SUPER^();
M_mapping();
IF sInstanceName='tote_1' THEN
	tote_status_array[0]	:= GVL.fb_loading.tote_status;
	tote_status_array[1]	:= GVL.fb_working1.tote_status;
	tote_status_array[2]	:= GVL.fb_working1.outboundTote_status;//outbound tote status form logtech
	machine_current_status	:= GVL.PackTags1.Status.StateCurrent;
	autostore_status		:= GVL.fb_autoStore1.autostore_status;
END_IF
IF sInstanceName='tote_2' THEN
	tote_status_array[0]	:= GVL.fb_loading.tote_status;
	tote_status_array[1]	:= GVL.fb_working2.tote_status;
	tote_status_array[2]	:= GVL.fb_working2.outboundTote_status;//outbound tote status form logtech
	machine_current_status	:= GVL.PackTags2.Status.StateCurrent;
	autostore_status		:= GVL.fb_autoStore2.autostore_status;
END_IF

CASE machine_current_status OF
	ePMLState_Aborted,ePMLState_Aborting:
		status	:= MachineStatus.ERROR;
	ePMLState_Stopping:	
		status	:= MachineStatus.STOPPING;
	ePMLState_Stopped:
		status	:= MachineStatus.STOPPED;
	ePMLState_Resetting:	
		status	:= MachineStatus.RESETTING;
	ePMLState_Idle:	
		status	:= MachineStatus.READY;		
	ePMLState_Execute:	
		status	:= MachineStatus.RUNNING;			
END_CASE

IF bInbound THEN
	inboundToteParams_temp.source_id	:= ModelIdentifier.inbounding_position;
	inboundToteParams_temp.target_id	:= ModelIdentifier.working_position;
	inbound_tote_request(inbound_tote_params:=inboundToteParams_temp);
	bInbound	:= FALSE;
END_IF
IF bOutbound THEN
	outboundToteParams_temp.source_id	:= ModelIdentifier.working_position;
	outboundToteParams_temp.target_id	:= ModelIdentifier.outbound_position;	
	outbound_tote_request(outbound_tote_params:=outboundToteParams_temp);
	bOutbound	:= FALSE;
END_IF
IF bAbortInbound THEN
	abortToreParams_temp.source_id	:= ModelIdentifier.inbounding_position;
	abortToreParams_temp.target_id	:= ModelIdentifier.working_position;	
	abort_tote_request(abort_tote_request_params:=abortToreParams_temp);
	bAbortInbound	:= FALSE;
END_IF

IF bAbortOutbound THEN
	abortToreParams_temp.source_id	:= ModelIdentifier.working_position;
	abortToreParams_temp.target_id	:= ModelIdentifier.outbound_position;	
	abort_tote_request(abort_tote_request_params:=abortToreParams_temp);
	bAbortOutbound	:= FALSE;
END_IF
IF bAutostore_exchange THEN
	autostore_control_command(Command:=AutostoreControlCommand.START);
	bAutostore_exchange	:= FALSE;
END_IF

{attribute 'TcRpcEnable'}
METHOD abort_tote_request : UDINT//only response while awaiting
VAR_INPUT
	abort_tote_request_params : AbortToteRequestParams; // Struct containing data from the barcode scan	
END_VAR
abort_tote_request:=MethodCallReturnValue.DECLINED_BUSY;
IF sInstanceName='tote_1' THEN
	IF abort_tote_request_params.source_id=ModelIdentifier.inbounding_position AND abort_tote_request_params.target_id=ModelIdentifier.working_position THEN
		iCase_abort	:= 1;
	END_IF
	IF abort_tote_request_params.source_id=ModelIdentifier.working_position AND abort_tote_request_params.target_id=ModelIdentifier.outbound_position THEN
		iCase_abort	:= 2;
	END_IF		
	CASE iCase_abort OF
		1:
			IF GVL.fb_working1.tote_status=ToteStatus.AWAITING_INBOUND_AVAILABILITY THEN
				subData.Topic	:= E_Topics.WORKING1_ABORT_INBOUND;
				GVL.PubSubService.Publish(topic:=E_Topics.WORKING1_ABORT_INBOUND,data:= subData);
				abort_tote_request:= MethodCallReturnValue.ACCEPTED;
			ELSE
				abort_tote_request:= MethodCallReturnValue.DECLINED_ERROR;
			END_IF
		2:
			IF GVL.fb_working1.tote_status=ToteStatus.AWAITING_OUTBOUND_AVAILABILITY THEN
				subData.Topic	:= E_Topics.WORKING1_ABORT_OUTBOUND;
				GVL.PubSubService.Publish(topic:=E_Topics.WORKING1_ABORT_OUTBOUND,data:= subData);
				abort_tote_request:= MethodCallReturnValue.ACCEPTED;
			ELSE
				abort_tote_request:= MethodCallReturnValue.DECLINED_ERROR;
			END_IF	
		ELSE
			abort_tote_request:= MethodCallReturnValue.DECLINED_ERROR;
	END_CASE
END_IF

IF sInstanceName='tote_2' THEN
	IF abort_tote_request_params.source_id=ModelIdentifier.inbounding_position AND abort_tote_request_params.target_id=ModelIdentifier.working_position THEN
		iCase_abort	:= 1;
	END_IF
	IF abort_tote_request_params.source_id=ModelIdentifier.working_position AND abort_tote_request_params.target_id=ModelIdentifier.outbound_position THEN
		iCase_abort	:= 2;
	END_IF		
	CASE iCase_abort OF
		1:
			IF GVL.fb_working2.tote_status=ToteStatus.AWAITING_INBOUND_AVAILABILITY THEN
				subData.Topic	:= E_Topics.WORKING2_ABORT_INBOUND;
				GVL.PubSubService.Publish(topic:=E_Topics.WORKING2_ABORT_INBOUND,data:= subData);
				abort_tote_request:= MethodCallReturnValue.ACCEPTED;
			ELSE
				abort_tote_request:= MethodCallReturnValue.DECLINED_ERROR;
			END_IF
		2:
			IF GVL.fb_working2.tote_status=ToteStatus.AWAITING_INBOUND_AVAILABILITY THEN
				subData.Topic	:= E_Topics.WORKING2_ABORT_OUTBOUND;
				GVL.PubSubService.Publish(topic:=E_Topics.WORKING2_ABORT_OUTBOUND,data:= subData);
				abort_tote_request:= MethodCallReturnValue.ACCEPTED;
			ELSE
				abort_tote_request:= MethodCallReturnValue.DECLINED_ERROR;
			END_IF	
		ELSE
			abort_tote_request:= MethodCallReturnValue.DECLINED_ERROR;			
	END_CASE
END_IF
END_METHOD

{attribute 'TcRpcEnable'}
METHOD autostore_control_command : BOOL
VAR_INPUT
	Command	: AutostoreControlCommand;
END_VAR
autostore_control_command	:= FALSE;
IF sInstanceName='tote_1' THEN
	subData.Topic	:= E_Topics.AUTOSTORE1_EXCHANGE;
	GVL.PubSubService.Publish(topic:= E_Topics.AUTOSTORE1_EXCHANGE,data:= subData);
END_IF
IF sInstanceName='tote_2' THEN
	subData.Topic	:= E_Topics.AUTOSTORE2_EXCHANGE;
	GVL.PubSubService.Publish(topic:= E_Topics.AUTOSTORE2_EXCHANGE,data:= subData);
END_IF
autostore_control_command	:= TRUE;
END_METHOD

{attribute 'TcRpcEnable'}
METHOD barcode_validation_request : UDINT
VAR_INPUT
	barcode_validation_request_params : BarcodeValidationRequestParams;
END_VAR
END_METHOD

{attribute 'TcRpcEnable'}
METHOD inbound_tote_request : UDINT
VAR_INPUT
	inbound_tote_params : InboundToteParams;
END_VAR
VAR	
	subData	: PubSubData;
END_VAR

IF sInstanceName='tote_1' THEN
//	IF NOT (((GVL.fb_working1.xLoading OR GVL.fb_working1.xInbound) AND GVL.fb_loading.xOutbound_woking1) OR 
//		GVL.fb_working1.tote_status=ToteStatus.LOADED OR GVL.fb_working1.xUnloading OR GVL.fb_working1.xOutbound) 
//	THEN//avoid cmd while inbounding or has tote
//		subData.Topic	:= E_Topics.WORKING1_INBOUND_TOTE;
//		GVL.PubSubService.Publish(topic:= E_Topics.WORKING1_INBOUND_TOTE,data:= subData);	
//	END_IF
	subData.Topic	:= E_Topics.WORKING1_INBOUND_TOTE;
	GVL.PubSubService.Publish(topic:= E_Topics.WORKING1_INBOUND_TOTE,data:= subData);
	A1	:= A1+1;	
END_IF
IF sInstanceName='tote_2' THEN
//	IF NOT (((GVL.fb_working2.xLoading OR GVL.fb_working2.xInbound) AND GVL.fb_loading.xOutbound_woking2) OR 
//		GVL.fb_working2.tote_status=ToteStatus.LOADED OR GVL.fb_working2.xUnloading OR GVL.fb_working2.xOutbound) 
//	THEN//avoid cmd while inbounding or has tote
//		subData.Topic	:= E_Topics.WORKING2_INBOUND_TOTE;
//		GVL.PubSubService.Publish(topic:= E_Topics.WORKING2_INBOUND_TOTE,data:= subData);
//	END_IF
	subData.Topic	:= E_Topics.WORKING2_INBOUND_TOTE;
	GVL.PubSubService.Publish(topic:= E_Topics.WORKING2_INBOUND_TOTE,data:= subData);
	A2	:= A2+1;
END_IF

//subData.Topic	:= E_Topics.RESET_WAITING_FOR_NEW_SPACE;
//GVL.PubSubService.Publish(topic:= E_Topics.RESET_WAITING_FOR_NEW_SPACE,data:= subData);
END_METHOD

{attribute 'TcRpcEnable'}
METHOD  init_tote_request : udint
VAR_INPUT
	init_tote_request_params : InitToteRequestParams;
END_VAR
init_tote_request:=1;
IF init_tote_request_params.source_id=ModelIdentifier.inbounding_position AND 
   init_tote_request_params.source_id=ModelIdentifier.working_position THEN 
  ;
     //MAIN.Machine.EM03.eState:=	E_WorkingStates.IDLE;				
//			MAIN.Machine.EM03.xLoading	:= FALSE;
//			MAIN.Machine.EM03.xUnloading	:= FALSE;
//			MAIN.Machine.EM03.xPerturbing := FALSE;
//			MAIN.Machine.EM03.xSwaping    := FALSE;
	 //MAIN.Machine.EM01.eState:=E_LoadingStates.IDLE;
END_IF  
IF init_tote_request_params.source_id=ModelIdentifier.working_position AND 
   init_tote_request_params.source_id=ModelIdentifier.outbound_position THEN 
;
    // MAIN.Machine.EM03.eState:=	E_WorkingStates.IDLE;				
//			MAIN.Machine.EM03.xLoading	:= FALSE;
//			MAIN.Machine.EM03.xUnloading	:= FALSE;
//			MAIN.Machine.EM03.xPerturbing := FALSE;
//			MAIN.Machine.EM03.xSwaping    := FALSE;
	// MAIN.Machine.EM04.eState:=E_UnloadingStates.IDLE;
END_IF  
init_tote_request:=0;
END_METHOD

METHOD M_mapping : BOOL
VAR_INPUT
END_VAR
END_METHOD

{attribute 'TcRpcEnable'}
METHOD outbound_tote_request : UDINT
VAR_INPUT
	outbound_tote_params : OutboundToteParams;	
END_VAR
VAR	
	subData	: PubSubData;
END_VAR
IF sInstanceName='tote_1' THEN
	IF NOT (GVL.fb_working1.xOutbound OR GVL.fb_working1.xInbound ) THEN//avoid cmd while outbounding
		subData.Topic	:= E_Topics.WORKING1_OUTBOUND_TOTE;
		GVL.PubSubService.Publish(topic:= E_Topics.WORKING1_OUTBOUND_TOTE,data:= subData);
	END_IF	
END_IF
IF sInstanceName='tote_2' THEN
	IF NOT (GVL.fb_working2.xOutbound OR GVL.fb_working2.xInbound ) THEN//avoid cmd while outbounding
		subData.Topic	:= E_Topics.WORKING2_OUTBOUND_TOTE;
		GVL.PubSubService.Publish(topic:= E_Topics.WORKING2_OUTBOUND_TOTE,data:= subData);
	END_IF
END_IF
END_METHOD

{attribute 'TcRpcEnable'}
METHOD perturb_tote_request : UDINT
VAR_INPUT
	perturb_tote_params : PerturbToteParams;	
END_VAR
IF //APP.Machine.CurrentStateEnum=E_PMLState.ePMLState_Execute 
//AND 
cmd=OrderToteCommand.DO_NOTHING
AND NOT MAIN.safety_1.bStop_button_unlock 
//AND NOT MAIN.safety_1.bBStop_button_unlock 
THEN
	cmd	:= OrderToteCommand.OPEN_BAG;
	perturb_tote_request:=0;
ELSE
	perturb_tote_request:=1;
END_IF
END_METHOD

{attribute 'TcRpcEnable'}
METHOD reset_tote_request : UDINT
VAR_INPUT
		
END_VAR
reset_tote_request	:= 1;

GVL.PackTags.Command.CntrlCmd:=1;

reset_tote_request	:= 0;
END_METHOD

{attribute 'TcRpcEnable'}
METHOD Setcmd : BOOL
VAR_INPUT
	orderToteCommand : OrderToteCommand;
END_VAR
cmd	:= orderToteCommand;
END_METHOD

{attribute 'TcRpcEnable'}
METHOD swap_tote_request : UDINT
VAR_INPUT
	swap_tote_params : SwapToteParams;	
END_VAR
IF //APP.Machine.CurrentStateEnum=E_PMLState.ePMLState_Execute 
//AND 
cmd=OrderToteCommand.DO_NOTHING
AND NOT MAIN.safety_1.bStop_button_unlock 
//AND NOT MAIN.safety_1.bBStop_button_unlock 
THEN
	cmd	:= OrderToteCommand.SWAP;
	swap_tote_request:=0;
ELSE
	swap_tote_request:=1;
END_IF
END_METHOD

END_FUNCTION_BLOCK

// ---- Mian/MAIN.TcPOU
// Disclaimer
// 
// This publication contains statements about the suitability of our products for certain areas of application. These statements are based on typical features of our products. The examples shown in this publication are for demonstration purposes only. 
// The information provided herein should not be regarded as specific operation characteristics. It is incumbent on the customer to check and decide whether a product is suitable for use in a particular application. 
// We do not give any warranty that the source code which is made available with this publication is complete or accurate. 
//
// THE SAMPLE CODE CONTAINED IN THIS PUBLICATION IS PROVIDED “AS IS” WITHOUT WARRANTY OF ANY KIND, EITHER EXPRESSED, IMPLIED OR STATUTORY, INCLUDING WITHOUT LIMITATION, ANY WARRANTY WITH RESPECT TO NON-INFRINGEMENT, FREEDOM FROM PROPRIETARY RIGHTS OF THIRD PARTIES OR FITNESS FOR ANY PARTICULAR PURPOSE. 
// This publication may be changed from time to time without prior notice. No liability is assumed for errors and/or omissions. Our products are described in detail in our data sheets and documentations. Product-specific warnings and cautions must be observed. 
// For the latest version of our data sheets and documentations visit our website (www.beckhoff.de). 
//
// © Beckhoff Automation GmbH & Co. KG, 2022
// The reproduction, distribution and utilization of this document as well as the communication of its contents to others without express authorization is prohibited. Offenders will be held liable for the payment of damages. All rights reserved in the event of the grant of a patent, utility model or design.
PROGRAM MAIN
VAR_INPUT
	bExecuteComplete			: BOOL;									//Command Execute Complete, not defined
END_VAR
VAR
	firstCycle : BOOL := TRUE;
	UserModeCofig				: PML_UnitModeConfig;					//User can configure his own Mode
	
	fbMachine					: FB_Machine;							//Instance of FB_Machine
//	fbMachine_2					: FB_Machine;							//Instance of FB_Machine
	bMachineStartedUp			: BOOL := FALSE;						//TRUE, when first PLC-Cycle finish
	fbVisu						: FB_Visu;								//Visualization
							//Visualization
	fbTrigger					: F_TRIG;								//Trigger for resseting Counters
	fbTrigger_2					: F_TRIG;								//Trigger for resseting Counters

	fbLocalSystemTime			 : FB_LocalSystemTime;					//Get local Systemtime
	fbLocalSystemTime_2			 : FB_LocalSystemTime;					//Get local Systemtime
	
	fbTriggerErrorMainAxis		: R_TRIG;								//Trigger for detecting Error on Mainaxis and write into PackTags
	fbTriggerErrorMetalAxis		: R_TRIG;								//Trigger for detecting Error on Metalaxis and write into PackTags
	fbTriggerErrorPlasticAxis	: R_TRIG;								//Trigger for detecting Error on Plasticaxis and write into PackTags
	
	nStateCommandCheck			: DINT;									//State to handle with statecommands
	
	i	: INT;

	FB_GetUPSStatus: FB_GetUPSStatus;	
	dataloaded: BOOL;								//UPS数据文件读取状态（True为读取成功，False为读取失败）
	OldData: BOOL;									//UPS备份数据文件读取状态
	PersistentDataStatus: EPlcPersistentStatus;		//Persistent数据读取（恢复）状态	
//	fb_ups	:FB_S_UPS_CX51x0;
	//application	: FB_Application;

	bButton				: BOOL;
	ton_button			: TON;

	refMachine_control_cmd	:REFERENCE TO MachineControlCommand;
	
	refMachine_control_cmd_2	:REFERENCE TO MachineControlCommand;
	
	rTrig_error	:ARRAY[0..10] OF R_TRIG;
	rTrig_error_2	:ARRAY[0..10] OF R_TRIG;
	
	rTrig_agingTest	:R_TRIG;
	fTrig_agingTest	:F_TRIG;

	topicCallbackTest	: E_Topics;
	dataCallbackTest	: PubSubData;
	topic_sample	: E_topic_sample;
	
	(***********************ADS********************************)
	light_tower_1			:	FB_Light_tower_module;
	light_tower_2			:	FB_Light_tower_module;
   // application_1			:	FB_Application;
	tote_1					:	FB_Tote_Subsystem;
	tote_2					:	FB_Tote_Subsystem;
	safety_1				:	FB_Safety_Subsystem;
	safety_2				:	FB_Safety_Subsystem;
	machine_control_1		:	FB_MachineControl_Subsystem;
	machine_control_2		:	FB_MachineControl_Subsystem;
	heartbeat_1				:	FB_HeartBeat_Subsystem;
	heartbeat_2				:	FB_HeartBeat_Subsystem;
	
	air_pressure_1			:	FB_AirPressure_Subsystem;
	air_pressure_2			:	FB_AirPressure_Subsystem;
	
	
	heartbeat_data_test : HeartbeatParams;	
	update_light_tower_params_test	: UpdateLightTowerParams;
	tset1: UDINT;
	
	
	version 				:	STRING(255);
	testbool: BOOL;
	inbound_tote_params_test : InboundToteParams;
	OutboundToteParams_test		:	OutboundToteParams;
	testbool1: BOOL;
	
	
	
	fbMachine1					: FB_Machine;							//Instance of FB_Machine
	fbMachine2					: FB_Machine;							//Instance of FB_Machine
	stateMachine1	: FB_StateMachine;
	stateMachine2	: FB_StateMachine;
	
	
END_VAR

(**************************************UPS*****************************************)
FB_GetUPSStatus(
	sNetId:= , 					//默认为本机Netid
	nPort:= , 					//ADS端口号，若不填写功能块会自动获取，默认0
	bEnable:= , 				//高电平有效，置True后循环读取UPS状态
	bValid=> , 					//当bValid为True时，stStatus的值有效
	bError=> , 
	nErrId=> , 
	stStatus=> );				//包含UPS信息的结构体
	

dataloaded:=_Appinfo.BootDataLoaded;
OldData:=_Appinfo.OldBootData;
PersistentDataStatus:=_Appinfo.PersistentStatus;

//application();
version:='v1.0.0';


//Call FB_Machine

GVL.fb_loading();
GVL.fb_working1();
GVL.fb_working2();
GVL.fb_autoStore1();
GVL.fb_autoStore2();
GVL.fb_working1._iModuleID:= ModuleID.WORKING1;
GVL.fb_working1._sInstanceName	:= 'working1';
GVL.fb_loading._iModuleID:= ModuleID.LOADING;
GVL.fb_loading._sInstanceName	:= 'loading';
GVL.fb_working2._iModuleID:= ModuleID.WORKING2;
GVL.fb_working2._sInstanceName	:= 'working2';
GVL.fb_autoStore1._sInstanceName	:= 'autoStore_1';
GVL.fb_autoStore1._iModuleID	:= ModuleID.AUTOSTORE1;
GVL.fb_autoStore2._sInstanceName	:= 'autoStore_2';
GVL.fb_autoStore2._iModuleID	:= ModuleID.AUTOSTORE2;

(***********************ADS********************************)
GVL.fb_mcp_1(id:=1);
heartbeat_1();
air_pressure_1(pPackTags:=ADR(GVL.PackTags1));
machine_control_1(pMachineCurrentStatus:= ADR(GVL.PackTags1.Status.StateCurrent));
tote_1();
safety_1(pHeartBeat:=ADR(heartbeat_1),pSafety_door:=ADR(GVL.fb_mcp_1.st_safety_door),pPackTags:=ADR(GVL.PackTags1),pMachine:=ADR(fbMachine1));
light_tower_1(pHeartBeat:=ADR(heartbeat_1),pLightTower:= ADR(GVL.fb_mcp_1.lightTower));

heartbeat_1._sInstanceName	:= 'heartBeat_1';
tote_1._sInstanceName	:='tote_1';
safety_1._sInstanceName	:='safety_1';
air_pressure_1._sInstanceName	:='air_pressure1';



GVL.fb_mcp_2(id:=2);
heartbeat_2();
air_pressure_2(pPackTags:=ADR(GVL.PackTags2));
machine_control_2(pMachineCurrentStatus:= ADR(GVL.PackTags2.Status.StateCurrent));
tote_2();
light_tower_2(pHeartBeat:=ADR(heartbeat_2),pLightTower:= ADR(GVL.fb_mcp_2.lightTower));
safety_2(pHeartBeat:=ADR(heartbeat_2),pSafety_door:=ADR(GVL.fb_mcp_2.st_safety_door),pPackTags:=ADR(GVL.PackTags2),pMachine:=ADR(fbMachine2));

heartbeat_1._sInstanceName	:= 'heartBeat_2';
tote_2._sInstanceName	:='tote_2';
safety_2._sInstanceName	:='safety_2';
air_pressure_2._sInstanceName	:='air_pressure2';





//Configure Usermode 1
A_UnitModeConfig();

//Runs the first PLC-Cycle
IF fbMachine1.bUndefinedDone AND fbMachine2.bUndefinedDone AND NOT bMachineStartedUp THEN
	GVL.PackTags1.Command.CntrlCmd	:= ePMLCommand_Abort;
	GVL.PackTags2.Command.CntrlCmd	:= ePMLCommand_Abort;
	bMachineStartedUp			:= TRUE;
END_IF


GVL.bButtonProductionReq := GVL.PackTags.Command.UnitMode = ePMLProtUnitMode_Production AND GVL.PackTags.Status.UnitModeCurrent <> GVL.PackTags.Command.UnitMode;

//Set the Packtags
M_SetPackTags();

//set the errors and warnings in Packtags
M_SetPackTagsErrorWarning();

//Call Visu
M_CallVisu();
///////////////////initialize unitmode and set 
IF GVL.PackTags.Command.UnitMode=ePMLProtUnitMode_Invalid THEN
	GVL.PackTags.Command.UnitMode	:= ePMLProtUnitMode_Production;
	GVL.PackTags.Command.Parameter[1].Value := 1;
	GVL.PackTags1.Command.UnitMode	:= ePMLProtUnitMode_Production;
	GVL.PackTags1.Command.Parameter[1].Value := 1;	
	GVL.PackTags2.Command.UnitMode	:= ePMLProtUnitMode_Production;
	GVL.PackTags2.Command.Parameter[1].Value := 1;	
	
END_IF


fbMachine1(	eModeCommand:= GVL.PackTags.Command.UnitMode,
  			eMode => GVL.PackTags1.Status.UnitModeCurrent, 
			eState =>GVL.PackTags1.Status.StateCurrent,
			pPML_Instance1:=ADR(GVL.fb_working1),
			pPML_Instance2:=ADR(GVL.fb_loading),
			pPackTags:=ADR(GVL.PackTags1),
			pSafetySystem	:= ADR(safety_1)
			);
			
fbMachine2(	eModeCommand:= GVL.PackTags.Command.UnitMode,
  			eMode => GVL.PackTags2.Status.UnitModeCurrent, 
			eState =>GVL.PackTags2.Status.StateCurrent,
			pPML_Instance1:=ADR(GVL.fb_working2),
			pPML_Instance2:=ADR(GVL.fb_loading),
			pPackTags:=ADR(GVL.PackTags2),
			pSafetySystem	:= ADR(safety_2)
			);		
	
stateMachine1(	pPackTags:=ADR(GVL.PackTags1),
				pMachine:=ADR(fbMachine1),
				pMachine_control_cmd := ADR(machine_control_1.machineControlCmd),
				pAirSystem	:=ADR(air_pressure_1),
				pSafetySystem	:= ADR(safety_1),
				pMcp	:= ADR(GVL.fb_mcp_1)
				);

stateMachine2(	pPackTags:=ADR(GVL.PackTags2),
				pMachine:=ADR(fbMachine2),
				pMachine_control_cmd := ADR(machine_control_2.machineControlCmd),
				pAirSystem	:=ADR(air_pressure_2),
				pSafetySystem	:= ADR(safety_2),
				pMcp	:= ADR(GVL.fb_mcp_2)
				);			
		
			
GVL.fbWriteLog(
	bWrite:= GVL.bWrite, 
	sFileName:= , 
	sMessage:= , 
	OK=> , 
	Busy=> , 
	ErrorMsg=> , 
	bError=> , 
	ErrorID=> );
	



M_SetUnitInfo();

ACTION A_UnitModeConfig:
UserModeCofig(
	eMode							:= ePMLUnitMode_Service, 
	bDisableClearing				:= TRUE, 
	bDisableStarting				:= FALSE, 
	bDisableSuspended				:= FALSE, 
	bDisableStopping				:= TRUE, 
	bDisableAborting				:= TRUE, 
	bDisableHolding					:= TRUE, 
	bDisableHeld					:= TRUE, 
	bDisableUnholding				:= TRUE, 
	bDisableSuspending				:= TRUE, 
	bDisableUnsuspending			:= TRUE, 
	bDisableResetting				:= TRUE, 
	bDisableIdle					:= FALSE, 
	bDisableCompleting				:= TRUE, 
	bDisableComplete				:= FALSE, 
	bEnableUnitModeChangeStopped	:= TRUE, 
	bEnableUnitModeChangeIdle		:= TRUE, 
	bEnableUnitModeChangeSuspended	:= FALSE, 
	bEnableUnitModeChangeExecute	:= FALSE, 
	bEnableUnitModeChangeAborted	:= TRUE, 
	bEnableUnitModeChangeHeld		:= FALSE, 
	bEnableUnitModeChangeComplete	:= TRUE, 
	bError							=> , 
	nErrorId						=> );
UserModeCofig(
	eMode							:= ePMLUnitMode_Production, 
	bDisableClearing				:= FALSE, 
	bDisableStarting				:= FALSE, 
	bDisableSuspended				:= TRUE, 
	bDisableStopping				:= FALSE, 
	bDisableAborting				:= FALSE, 
	bDisableHolding					:= TRUE, 
	bDisableHeld					:= TRUE, 
	bDisableUnholding				:= TRUE, 
	bDisableSuspending				:= TRUE, 
	bDisableUnsuspending			:= TRUE, 
	bDisableResetting				:= FALSE, 
	bDisableIdle					:= FALSE, 
	bDisableCompleting				:= FALSE, 
	bDisableComplete				:= FALSE, 
	bEnableUnitModeChangeStopped	:= TRUE, 
	bEnableUnitModeChangeIdle		:= TRUE, 
	bEnableUnitModeChangeSuspended	:= FALSE, 
	bEnableUnitModeChangeExecute	:= FALSE, 
	bEnableUnitModeChangeAborted	:= TRUE, 
	bEnableUnitModeChangeHeld		:= FALSE, 
	bEnableUnitModeChangeComplete	:= TRUE, 
	bError							=> , 
	nErrorId						=> );
END_ACTION

METHOD M_CallVisu
VAR_INPUT
END_VAR
//Calling FB_Visu
fbVisu(
	aKeyPressed				:= GVL.aKeyPressed,
	aUnitInfo				:= GVL.aUnitInfo, 
	bInvalidEntry			=> ,
	aCaption				=> GVL.aCaption,
	eModeVisu				=> ,
	eStateVisu				=> ,
	sUnitName				=> ,
	iFrameVisible			=> );
END_METHOD

METHOD M_SetPackTags
VAR_INPUT
END_VAR
VAR	
END_VAR
//***************************Writing Data into GVL.PackTags***************************

//Parameters for the production
GVL.PackTags.Command.Parameter[1].ID				:= 1;
GVL.PackTags.Command.Parameter[1].Name				:= 'Quantity';
GVL.PackTags.Command.Parameter[1].Unit				:= 'Tote';

//Countig produced totes, see fb_sample1
GVL.PackTags.Admin.ProdProcessedCount[1].ID			:= 1;
GVL.PackTags.Admin.ProdProcessedCount[1].Name		:= 'ToteFinish_Sample';
GVL.PackTags.Admin.ProdProcessedCount[1].Unit		:= 'Tote';





//Write the actual state and mode into the GVL.PackTags
GVL.PackTags.Status.StateCurrent					:= fbMachine1.eState;
GVL.PackTags.Status.UnitModeCurrent					:= fbMachine1.eMode;
GVL.PackTags.Status.StateRequested					:= fbMachine1.eCommand;
GVL.PackTags.Status.UnitModeRequested				:= fbMachine1.eModeCommand;
GVL.PackTags.Status.StateChangeInProcess			:= GVL.PackTags.Status.StateCurrent <> GVL.PackTags.Status.StateRequested;
GVL.PackTags.Status.UnitModeChangeInProcess			:= GVL.PackTags.Status.UnitModeCurrent <> GVL.PackTags.Status.UnitModeRequested;

//Write the actual state and mode into the GVL.PackTags2
GVL.PackTags1.Status.StateCurrent					:= fbMachine1.eState;
GVL.PackTags1.Status.UnitModeCurrent					:= fbMachine1.eMode;
GVL.PackTags1.Status.StateRequested					:= fbMachine1.eCommand;
GVL.PackTags1.Status.UnitModeRequested				:= fbMachine1.eModeCommand;
GVL.PackTags1.Status.StateChangeInProcess			:= GVL.PackTags1.Status.StateCurrent <> GVL.PackTags1.Status.StateRequested;
GVL.PackTags1.Status.UnitModeChangeInProcess			:= GVL.PackTags1.Status.UnitModeCurrent <> GVL.PackTags1.Status.UnitModeRequested;
//Write the actual state and mode into the GVL.PackTags2
GVL.PackTags2.Status.StateCurrent					:= fbMachine2.eState;
GVL.PackTags2.Status.UnitModeCurrent					:= fbMachine2.eMode;
GVL.PackTags2.Status.StateRequested					:= fbMachine2.eCommand;
GVL.PackTags2.Status.UnitModeRequested				:= fbMachine2.eModeCommand;
GVL.PackTags2.Status.StateChangeInProcess			:= GVL.PackTags2.Status.StateCurrent <> GVL.PackTags2.Status.StateRequested;
GVL.PackTags2.Status.UnitModeChangeInProcess			:= GVL.PackTags2.Status.UnitModeCurrent <> GVL.PackTags2.Status.UnitModeRequested;


//Write actual time and date in GVL.PackTags
fbLocalSystemTime(sNetID:= '', bEnable := TRUE);
GVL.PackTags.Admin.PlcDateTime[0]	:= fbLocalSystemTime.systemTime.wYear;
GVL.PackTags.Admin.PlcDateTime[1]	:= fbLocalSystemTime.systemTime.wMonth;
GVL.PackTags.Admin.PlcDateTime[2]	:= fbLocalSystemTime.systemTime.wDay;
GVL.PackTags.Admin.PlcDateTime[3]	:= fbLocalSystemTime.systemTime.wHour;
GVL.PackTags.Admin.PlcDateTime[4]	:= fbLocalSystemTime.systemTime.wMinute;
GVL.PackTags.Admin.PlcDateTime[5]	:= fbLocalSystemTime.systemTime.wSecond;
GVL.PackTags.Admin.PlcDateTime[6]	:= fbLocalSystemTime.systemTime.wMilliseconds;
GVL.PackTags1.Admin.PlcDateTime	:= GVL.PackTags.Admin.PlcDateTime;
GVL.PackTags2.Admin.PlcDateTime	:= GVL.PackTags.Admin.PlcDateTime;
//Set the productcounter to 0, when the production command is completed
fbTrigger(CLK:= (fbMachine1.eState = ePMLState_Complete));
IF fbTrigger.Q OR GVL.stChangeIntoProduction.bYesReset THEN
	GVL.PackTags1.Admin.ProdProcessedCount[1].Count	:= 0;
	GVL.PackTags1.Command.Parameter[1].Value			:= 0;
	GVL.nVisuProductCommand							:= 0;
END_IF

//Set the productcounter to 0, when the production command is completed
fbTrigger(CLK:= (fbMachine2.eState = ePMLState_Complete));
IF fbTrigger.Q OR GVL.stChangeIntoProduction.bYesReset THEN
	GVL.PackTags2.Admin.ProdProcessedCount[1].Count	:= 0;
	GVL.PackTags2.Command.Parameter[1].Value			:= 0;
	GVL.nVisuProductCommand							:= 0;
END_IF
END_METHOD

METHOD M_SetPackTagsErrorWarning
VAR_INPUT
END_VAR
//====================Error and Warnig setting========================
//Warnings
GVL.PackTags1.Admin.Warning[1].Message	:= 'Invalid Production Command, command Products must be higher than 0';
GVL.PackTags1.Admin.Warning[1].ID 		:= 1;

GVL.PackTags1.Admin.Warning[2].Message	:= 'Invalid Mode Command, please try anothereone';
GVL.PackTags1.Admin.Warning[2].ID		:= 2;


//====================Error and Warnig handling========================
//warning for invalid production command
IF 	GVL.PackTags1.Status.UnitModeCurrent = ePMLProtUnitMode_Production AND 
	GVL.PackTags1.Status.StateCurrent = ePMLState_Idle AND 
	GVL.PackTags1.Command.CntrlCmd = ePMLCommand_Start AND
 	GVL.PackTags1.Command.Parameter[1].Value <= 0 
THEN
	GVL.PackTags1.Admin.Warning[1].Trigger :=TRUE;
ELSE
	GVL.PackTags1.Admin.Warning[1].Trigger :=FALSE;
END_IF

//warning for invalid mode command
IF fbMachine1.bInvalidModeCommandOut THEN
	GVL.PackTags1.Admin.Warning[2].Trigger :=TRUE;
ELSE 
	GVL.PackTags1.Admin.Warning[2].Trigger :=FALSE;
END_IF





//====================Error and Warnig setting========================
//Warnings
GVL.PackTags1.Admin.Warning[1].Message	:= 'Invalid Production Command, command Products must be higher than 0';
GVL.PackTags1.Admin.Warning[1].ID 		:= 1;

GVL.PackTags1.Admin.Warning[2].Message	:= 'Invalid Mode Command, please try anothereone';
GVL.PackTags1.Admin.Warning[2].ID		:= 2;


//====================Error and Warnig handling========================
//warning for invalid production command
IF 	GVL.PackTags2.Status.UnitModeCurrent = ePMLProtUnitMode_Production AND 
	GVL.PackTags2.Status.StateCurrent = ePMLState_Idle AND 
	GVL.PackTags2.Command.CntrlCmd = ePMLCommand_Start AND
 	GVL.PackTags2.Command.Parameter[1].Value <= 0 
THEN
	GVL.PackTags2.Admin.Warning[1].Trigger :=TRUE;
ELSE
	GVL.PackTags2.Admin.Warning[1].Trigger :=FALSE;
END_IF

//warning for invalid mode command
IF fbMachine2.bInvalidModeCommandOut THEN
	GVL.PackTags2.Admin.Warning[2].Trigger :=TRUE;
ELSE 
	GVL.PackTags2.Admin.Warning[2].Trigger :=FALSE;
END_IF
END_METHOD

METHOD M_SetUnitInfo
VAR_INPUT
END_VAR
GVL.aUnitInfo[eMachine1].Name			:= 'fbMachine1';
GVL.aUnitInfo[eMachine1].ActMode			:= fbMachine1.eMode;
GVL.aUnitInfo[eMachine1].ActState		:= fbMachine1.eState;

GVL.aUnitInfo[eMachine1].Name			:= 'fbMachine2';
GVL.aUnitInfo[eMachine1].ActMode		:= fbMachine2.eMode;
GVL.aUnitInfo[eMachine1].ActState		:= fbMachine2.eState;

//GVL.aUnitInfo[eSample].Name				:= GVL.fb_sample._sInstanceName;
//GVL.aUnitInfo[eSample].ActMode			:= GVL.fb_sample.eMode;
//GVL.aUnitInfo[eSample].ActState			:= GVL.fb_sample.eState;


GVL.aUnitInfo[eLoading].Name			:= GVL.fb_loading._sInstanceName;
GVL.aUnitInfo[eLoading].ActMode			:= GVL.fb_loading.eMode;
GVL.aUnitInfo[eLoading].ActState		:= GVL.fb_loading.eState;


GVL.aUnitInfo[eWorking1].Name			:= GVL.fb_working1._sInstanceName;
GVL.aUnitInfo[eWorking1].ActMode		:= GVL.fb_working1.eMode;
GVL.aUnitInfo[eWorking1].ActState		:= GVL.fb_working1.eState;


GVL.aUnitInfo[eWorking2].Name			:= GVL.fb_working2._sInstanceName;
GVL.aUnitInfo[eWorking2].ActMode		:= GVL.fb_working2.eMode;
GVL.aUnitInfo[eWorking2].ActState		:= GVL.fb_working2.eState;
END_METHOD

END_PROGRAM

// ---- Mian/FB_StateMachine.TcPOU
FUNCTION_BLOCK FB_StateMachine
VAR_INPUT
	
	pPackTags				: POINTER TO ST_PackMLv30;
	pMachine				: POINTER TO FB_Machine;	
	pMachine_control_cmd	: POINTER TO MachineCommandStructure;	
	pAirSystem				: POINTER TO FB_AirPressure_Subsystem;
	pSafetySystem			: POINTER TO FB_Safety_Subsystem;	
	pMcp					: POINTER TO FB_mcp;
END_VAR
VAR_OUTPUT
END_VAR
VAR
	rTrig_error	:ARRAY[1..10] OF R_TRIG;
	i	: INT;
		

END_VAR

(*command from 1:PLC HMI buttons;2:APP;3:Safety module;4:each modules*)
/////////////////////////////abort/////////////////////////////	
IF 	pMachine^.eState <> ePMLState_Aborted AND pMachine^.eState <> ePMLState_Clearing THEN	
	IF pPackTags^.Command.CntrlCmd = ePMLCommand_Abort OR M_CheckError() THEN
		IF pMachine^.M_UnitsActive(ePMLCommand_Abort) THEN
			pMachine^.eCommand	:= ePMLCommand_Abort;
			pMachine_control_cmd^.command	:= MachineControlCommand.DO_NOTHING;
		END_IF
	END_IF
END_IF
/////////////////////////////stop/////////////////////////////
IF M_CheckError() THEN
	//
ELSE					
	IF (pPackTags^.Command.CntrlCmd = ePMLCommand_Stop OR 
		pMachine_control_cmd^.command = MachineControlCommand.STOP OR 
		pSafetySystem^.pml_command=ePMLCommand_Stop) AND pMachine^.eState <> ePMLState_Stopped
	THEN
		IF pMachine^.M_UnitsActive(ePMLCommand_Stop) THEN
			pMachine^.eCommand	:= ePMLCommand_Stop;
		END_IF
	END_IF
END_IF

CASE pMachine^.eState OF
			
	ePMLState_Aborted:
		IF pMcp^.st_safety_door.button_reset THEN
			pPackTags^.Command.CntrlCmd := ePMLCommand_Clear;
		END_IF
		IF 	pPackTags^.Command.CntrlCmd = ePMLCommand_Clear OR
			(pSafetySystem^.safety_status=SafetyStatus.READY AND pMachine_control_cmd^.command=MachineControlCommand.RESET)//while safety is ready,can be reset remotely	 
		THEN
			IF pSafetySystem^.M_reset() THEN	//reset safety first
				IF pSafetySystem^.xError THEN
					pPackTags^.Command.CntrlCmd		:= ePMLCommand_Undefined;
					pMachine_control_cmd^.command	:= MachineControlCommand.DO_NOTHING;
				ELSE
					IF pMachine^.M_UnitsActive(ePMLCommand_Clear) THEN
						pMachine^.eCommand	:= ePMLCommand_Clear;
					END_IF					
				END_IF
			END_IF	
		END_IF
		//reset command
		IF pMachine^.eCommand = ePMLCommand_Abort THEN
			pMachine^.eCommand	:= ePMLCommand_Undefined;
		END_IF
			
	ePMLState_Complete:		
		IF (pPackTags^.Command.CntrlCmd = ePMLCommand_Reset OR pMachine_control_cmd^.command = MachineControlCommand.RESET (*OR
		 	pMcp^.st_safety_door.button_reset*)) 
		THEN
			pMachine^.eCommand	:= ePMLCommand_Reset;
		END_IF
			
			
	ePMLState_Idle:
		IF (pPackTags^.Command.CntrlCmd = ePMLCommand_Start OR pMachine_control_cmd^.command = MachineControlCommand.START)	AND
			(NOT (pPackTags^.Command.Parameter[1].Value <= 0) OR NOT (pMachine^.eMode = 1))
		THEN	
			IF pMachine^.M_UnitsActive(ePMLCommand_Start) THEN
				pMachine^.eCommand	:= ePMLCommand_Start;
			END_IF
		END_IF
		IF pMachine_control_cmd^.command = MachineControlCommand.RESET THEN
			pMachine_control_cmd^.command	:= MachineControlCommand.DO_NOTHING;
		END_IF
		//reset command
		IF pMachine^.eCommand = ePMLCommand_Reset THEN
			pMachine^.eCommand	:= ePMLCommand_Undefined;
		END_IF
			
			
	ePMLState_Stopped:
		IF pPackTags^.Command.CntrlCmd = ePMLCommand_Reset OR pMachine_control_cmd^.command = MachineControlCommand.RESET THEN		
			IF pMachine^.M_UnitsActive(ePMLCommand_Reset) THEN
				pMachine^.eCommand	:= ePMLCommand_Reset;
			END_IF
		END_IF		
		IF (pPackTags^.Command.CntrlCmd = ePMLCommand_Start OR pMachine_control_cmd^.command = MachineControlCommand.START)	AND
			(NOT (pPackTags^.Command.Parameter[1].Value <= 0) OR NOT (pMachine^.eMode = 1)) AND
			stPMLUnitModeConfiguration[pMachine^.eMode].aStateDisabled[ePMLState_Idle] 
		THEN	
			IF pMachine^.M_UnitsActive(ePMLCommand_Start) THEN
				pMachine^.eCommand	:= ePMLCommand_Start; 	
			END_IF			
		END_IF	
		IF pMachine_control_cmd^.command = MachineControlCommand.STOP THEN
			pMachine_control_cmd^.command	:= MachineControlCommand.DO_NOTHING;
		END_IF	
		//reset command
		IF pMachine^.eCommand = ePMLCommand_Clear OR pMachine^.eCommand = ePMLCommand_Stop THEN
			pMachine^.eCommand	:= ePMLCommand_Undefined;
		END_IF
			
			
	ePMLState_Execute:	
		IF pMachine_control_cmd^.command = MachineControlCommand.START THEN
			pMachine_control_cmd^.command	:= MachineControlCommand.DO_NOTHING;
		END_IF
		IF pPackTags^.Command.CntrlCmd = ePMLCommand_Hold	AND	
			(pMachine^.eMode =  1 OR pMachine^.eMode =  4 OR pMachine^.eMode = 2)  
		THEN
			pMachine^.eCommand	:= ePMLCommand_Hold;
		END_IF	
		IF pPackTags^.Command.CntrlCmd = ePMLCommand_Suspend AND (pMachine^.eMode = 4 OR pMachine^.eMode = 1)THEN
		 
			pMachine^.eCommand	:= ePMLCommand_Suspend;
		END_IF	 
		//reset command
		IF pMachine^.eCommand = ePMLCommand_Start THEN
			pMachine^.eCommand	:= ePMLCommand_Undefined;
		END_IF
			
			
	ePMLState_Held:	 
		IF pPackTags^.Command.CntrlCmd = ePMLCommand_Unhold THEN
			pMachine^.eCommand	:= ePMLCommand_Unhold;
		END_IF
			
			
	ePMLState_Suspended:
		IF pPackTags^.Command.CntrlCmd = ePMLCommand_Unsuspend THEN
			pMachine^.eCommand	:= ePMLCommand_Unsuspend;
		END_IF
			
			
	ePMLState_Aborting,ePMLState_Clearing,ePMLState_Resetting,ePMLState_Starting,ePMLState_Stopping:
		pPackTags^.Command.CntrlCmd	:= ePMLCommand_Undefined;

		
		
END_CASE

METHOD M_CheckError : BOOL

VAR
	
END_VAR
M_CheckError	:= FALSE;

FOR i:=1 TO GlobalParameters.MaxAlarms DO
	IF pPackTags^.Admin.Alarm[i].Trigger THEN
		M_CheckError	:= TRUE;
	END_IF
END_FOR
//RETURN;//remove this while safety and air is ready
IF pSafetySystem^.xError OR pAirSystem^.xError THEN
	M_CheckError	:= TRUE;
END_IF
END_METHOD

END_FUNCTION_BLOCK

// ---- Mian/FB_loading_tote.TcPOU
FUNCTION_BLOCK FB_loading_tote EXTENDS FB_Generic
VAR_INPUT

END_VAR
VAR_OUTPUT
	
END_VAR
VAR
	eStates			: E_LoadingStates := E_LoadingStates.IDLE;
	eStateTemp		: E_LoadingStates := E_LoadingStates.IDLE;
	eTransfer			: E_Transfer;
//	current_tote_status	: ToteStatus;
	tote_status	: ToteStatus;
	
///////////////hardware define//////////////////
	roller_assign : Roller_x;         //X-Belt
	roller_inbound: Roller_y;         //Y向滚筒1
	roller_inbound_assist:Roller_y;   //Y向滚筒2
	valve_left_door:Valve;
    valve_right_door:Valve;
	
	limit_sensor_positive:BOOL;
    limit_sensor_negative:BOOL;
    limit_sensor_home:BOOL;

	
	rRight_Door_Extend		: R_TRIG;
	
	rLeft_Door_Extend		: R_TRIG;
	
	rRight_Door_Retract		: R_TRIG;
	
	rLeft_Door_Retract		: R_TRIG;
	//photo_sensor_tote_detection	: FB_DigitalInput;
	photo_sensor_diagonal       : FB_DigitalInput;  
    photo_sensor_bottom         : FB_DigitalInput;
	
	bLoadingLeft: BOOL;
	bLoadingRight: BOOL;
	
	EDM_KM						: BOOL;
	floodlight					: BOOL;
	mcAxis	 					: FB_MotionAxis_MC;
	st_mcAxis					: ST_MotionAxis_MC;
	AxisRef						: AXIS_REF;	
	D: INT;
	on_ms: INT;
	off_ms: INT;
	bTest: BOOL;
	xOutbound_woking1			: BOOL;//from cmd of app
	xBeginOutbound_Working1		: BOOL;
	xEndOutbound_Working1		: BOOL;
	
	
	xOutbound_woking2			: BOOL;//from cmd of app
	xBeginOutbound_Working2		: BOOL;
	xEndOutbound_Working2		: BOOL;
	
	logtech_load_command	: LogTechControlCmd;
	logtech_load_status		: LogTechTransferStatus;
	byteIn	AT%I* : ARRAY [0..15] OF BYTE;//[0]:transfer status;[1]:heart_ beat;[2]:logtech station status;[3]:logtech_load_status
	byteOut	AT%Q* : ARRAY [0..15] OF BYTE;//[0]:transfer command;[1]:heart_beat;[2]:Covariant station status;[3]:logtech_load_command
	

	responsing_unlock1	: BOOL;
	responsing_unlock2	: BOOL;
	xLocking1	: BOOL;
	xLocking2	: BOOL;
	xUnlocking1	: BOOL;
	xUnlocking2	: BOOL;
END_VAR

VAR CONSTANT
	rMax_lift	: REAL	:= 800;
	rMin_lift	: REAL	:= -1;
END_VAR

VAR PERSISTENT
	rPos_load	: REAL;
	rPos_unload	: REAL;	
END_VAR

SUPER^();
IF NOT subscribed THEN
	GVL.PubSubService.Subscribe(E_Topics.WORKING1_INBOUND_TOTE,sInstanceName,THIS^);
	GVL.PubSubService.Subscribe(E_Topics.LOADING_BEGIN_OUTBOUND_WOKING1,sInstanceName,THIS^);
	GVL.PubSubService.Subscribe(E_Topics.LOADING_END_OUTBOUND_WOKING1,sInstanceName,THIS^);
	GVL.PubSubService.Subscribe(E_Topics.WORKING1_ABORT_INBOUND,sInstanceName,THIS^);
	GVL.PubSubService.Subscribe(E_Topics.WORKING2_INBOUND_TOTE,sInstanceName,THIS^);
	GVL.PubSubService.Subscribe(E_Topics.LOADING_BEGIN_OUTBOUND_WOKING2,sInstanceName,THIS^);
	GVL.PubSubService.Subscribe(E_Topics.LOADING_END_OUTBOUND_WOKING2,sInstanceName,THIS^);	
	GVL.PubSubService.Subscribe(E_Topics.RESET_WAITING_FOR_NEW_SPACE,sInstanceName,THIS^);
	GVL.PubSubService.Subscribe(E_Topics.WORKING2_ABORT_INBOUND,sInstanceName,THIS^);
	subscribed	:= TRUE;
END_IF

infoLevel	:= ServerityLevelType.WARNING;


////////////////////////////////////////////////electrical error///////////////////////////////////////////////////
rTrig_electricalError[1](CLK:= st_mcAxis.mcReadStatus.Error);
rTrig_electricalError[2](CLK:= roller_assign.roller.err.Q);
rTrig_electricalError[3](CLK:= roller_inbound.roller.err.Q);
//rTrig_electricalError[4](CLK:= roller_inbound_assist.roller.err.Q);
IF GVL.PackTags.Status.StateCurrent<>E_PMLState.ePMLState_Resetting THEN
	FOR i:=1 TO 10 DO
		IF rTrig_electricalError[i].Q THEN
			THIS^.packTags.Admin.Alarm[i].ID	:= i;
			CASE i OF
				1:
					THIS^.packTags.Admin.Alarm[1].Message	:= GenerateErrorMsg(errorType:='E',iState := i,errorMsg:='axis is in error state.');
				2:
					THIS^.packTags.Admin.Alarm[2].Message	:= GenerateErrorMsg(errorType:='E',iState := i,errorMsg:='assign roller is in error state.');
				3:
					THIS^.packTags.Admin.Alarm[3].Message	:= GenerateErrorMsg(errorType:='E',iState := i,errorMsg:='inbound roller is in error state.');
				4:
					THIS^.packTags.Admin.Alarm[4].Message	:= GenerateErrorMsg(errorType:='E',iState := i,errorMsg:='inbound assist roller is in error state.');
			END_CASE
			tote_status	:= ToteStatus.ELECTRICAL_ERROR;
			GVL.pml_adminAlarm.M_SetAlarm(stAdmin:=GVL.PackTags1.Admin,stAlarm := THIS^.packTags.Admin.Alarm[i]);
			GVL.pml_adminAlarm.M_SetAlarm(stAdmin:=GVL.PackTags2.Admin,stAlarm := THIS^.packTags.Admin.Alarm[i]);
			isError	:= TRUE;
		END_IF
	END_FOR
END_IF

(*
Description: 
the callback that will be invoked when there is a publish for what the subscriber was subscribed to.
*)
METHOD Callback
VAR_INPUT
	data : PubSubData;
END_VAR
CASE data.Topic OF
	E_Topics.WORKING1_INBOUND_TOTE:
		IF NOT xOutbound_woking1 AND GVL.fb_working1.tote_status<>ToteStatus.LOADED THEN
			xOutbound_woking1	:= TRUE;
		END_IF
		
//	E_Topics.LOADING_BEGIN_OUTBOUND_WOKING1:
//		xBeginOutbound_Working1	:= TRUE;
	E_Topics.LOADING_END_OUTBOUND_WOKING1:
		xOutbound_woking1	:= FALSE;
		xBeginOutbound_Working1	:= FALSE;
		xEndOutbound_Working1	:= TRUE;	
		
	E_Topics.WORKING2_INBOUND_TOTE:
		IF NOT xOutbound_woking2 AND GVL.fb_working2.tote_status<>ToteStatus.LOADED THEN 
			xOutbound_woking2	:= TRUE;
		END_IF
//	E_Topics.LOADING_BEGIN_OUTBOUND_WOKING2:
//		xBeginOutbound_Working2	:= TRUE;
	E_Topics.LOADING_END_OUTBOUND_WOKING2:
		xOutbound_woking2	:= FALSE;
		xBeginOutbound_Working2	:= FALSE;
		xEndOutbound_Working2	:= TRUE;
	E_Topics.RESET_WAITING_FOR_NEW_SPACE:
		ton_timeout.IN	:= FALSE;
	E_Topics.WORKING1_ABORT_INBOUND:
		xOutbound_woking1	:= FALSE;
	E_Topics.WORKING2_ABORT_INBOUND:
		xOutbound_woking2	:= FALSE;
END_CASE
END_METHOD

{attribute 'object_name' := 'M_Aborting'}
METHOD M_Aborting
CASE fbUnitModeManager.eModeStatus OF	
	ePMLProtUnitMode_Production, ePMLProtUnitMode_Manual:		
		roller_assign.roller.forward := FALSE;
		roller_assign.roller.backward := FALSE;
		roller_inbound.roller.forward := FALSE;
		roller_inbound.roller.backward := FALSE;
		roller_inbound_assist.roller.forward := FALSE;
		roller_inbound_assist.roller.backward := FALSE;
		st_mcAxis.mcMoveAbsolute.Execute	:= FALSE;
		st_mcAxis.mcStop.Execute	:= TRUE;	
		xOutbound_woking1	:= FALSE;
		xOutbound_woking2	:= FALSE;
		bAging_test	:= FALSE;
		iAging_test	:= 0;
		M_StateComplete();
			
	ePMLProtUnitMode_Maintenance, ePMLUnitMode_Service:
		
		M_StateComplete();
END_CASE
END_METHOD

METHOD M_agingTest : BOOL
VAR_INPUT
	rVelocity_percent	: REAL;
END_VAR
ton_aging_test();
CASE iAging_test OF
	0://
	
	1://run forward
		ton_aging_test.PT	:= T#5S;
		ton_aging_test.IN	:= TRUE;
		st_mcAxis.mcMoveAbsolute.Execute	:= TRUE;						
		st_mcAxis.rActualPosSet	:= rPos_load;
		st_mcAxis.rVelocitySet	:= rVelocity_percent*300;
		roller_assign.roller.forward	:= TRUE;
		roller_inbound.roller.forward	:= TRUE;
		roller_inbound_assist.roller.forward	:= TRUE;
		valve_left_door.extend 		:= TRUE;
		valve_left_door.retract		:= FALSE;
		valve_right_door.extend 	:= TRUE;
		valve_right_door.retract	:= FALSE;		
		IF st_mcAxis.mcMoveAbsolute.Done AND valve_left_door.extended AND NOT valve_left_door.retracted AND valve_right_door.extended AND NOT valve_right_door.retracted THEN
			st_mcAxis.mcMoveAbsolute.Execute	:= FALSE;
			roller_assign.roller.forward	:= FALSE;
			roller_inbound.roller.forward	:= FALSE;
			roller_inbound_assist.roller.forward	:= FALSE;
			ton_aging_test.IN	:= FALSE;			
			iAging_test	:= 2;
		END_IF	
	2:	
		ton_aging_test.PT	:= T#3S;
		ton_aging_test.IN	:= TRUE;
		IF ton_aging_test.Q THEN
			ton_aging_test.IN	:= FALSE;
			iAging_test	:= 3;				
		END_IF
	3://run backward
		ton_aging_test.PT	:= T#5S;
		ton_aging_test.IN	:= TRUE;
		st_mcAxis.mcMoveAbsolute.Execute	:= TRUE;						
		st_mcAxis.rActualPosSet	:= rPos_unload;
		st_mcAxis.rVelocitySet	:= rVelocity_percent*300;
		roller_assign.roller.backward	:= TRUE;
		roller_inbound.roller.forward	:= TRUE;
		roller_inbound.roller.backward	:= TRUE;
		roller_inbound_assist.roller.forward	:= TRUE;
		roller_inbound_assist.roller.backward	:= TRUE;
		valve_left_door.extend 		:= FALSE;
		valve_left_door.retract		:= TRUE;
		valve_right_door.extend 	:= FALSE;
		valve_right_door.retract	:= TRUE;		
		IF st_mcAxis.mcMoveAbsolute.Done AND NOT valve_left_door.extended AND valve_left_door.retracted AND NOT valve_right_door.extended AND valve_right_door.retracted THEN
			st_mcAxis.mcMoveAbsolute.Execute	:= FALSE;
			roller_assign.roller.backward	:= FALSE;
			roller_inbound.roller.forward	:= FALSE;
			roller_inbound.roller.backward	:= FALSE;
			roller_inbound_assist.roller.forward	:= FALSE;
			roller_inbound_assist.roller.backward	:= FALSE;	
			ton_aging_test.IN	:= FALSE;			
			iAging_test	:= 4;
		END_IF	
	4:
		ton_aging_test.PT	:= T#3S;
		ton_aging_test.IN	:= TRUE;
		IF ton_aging_test.Q THEN
			diCnt_aging	:= diCnt_aging+1;
			ton_aging_test.IN	:= FALSE;
			ADSLOGSTR(msgCtrlMask:=Tc2_System.ADSLOG_MSGTYPE_LOG,msgFmtStr:=CONCAT(STR1:=sInstanceName,STR2:=DINT_TO_STRING(diCnt_aging)),strArg:='');
			iAging_test	:= 1;				
		END_IF
	
		
		
		
	10://stop
		st_mcAxis.mcMoveAbsolute.Execute	:= FALSE;
		roller_assign.roller.forward	:= FALSE;
		roller_assign.roller.backward	:= FALSE;
		roller_inbound.roller.forward	:= FALSE;	
		roller_inbound.roller.backward	:= FALSE;
		roller_inbound_assist.roller.forward	:= FALSE;
		roller_inbound_assist.roller.backward	:= FALSE;		
		valve_left_door.extend 		:= FALSE;
		valve_left_door.retract		:= TRUE;
		valve_right_door.extend 	:= FALSE;
		valve_right_door.retract	:= TRUE;
		ton_aging_test.IN	:= FALSE;		
		iAging_test	:= 0;

	END_CASE
END_METHOD

{attribute 'object_name' := 'M_Completing'}
METHOD M_Completing
CASE fbUnitModeManager.eModeStatus OF
	ePMLProtUnitMode_Production:
		;
END_CASE
END_METHOD

{attribute 'object_name' := 'M_Execute'}
METHOD M_Execute

VAR

	
END_VAR
CASE fbUnitModeManager.eModeStatus OF
	ePMLProtUnitMode_Production:		//Mode Production

//////////////////////////////////////////////////////////timeout//////////////////////////////////////////
		iStateTemp	:= eStateTemp;
//		ton_timeout();
		IF eStateTemp=eStates THEN
			ton_timeout.IN	:=TRUE;
		ELSE
			ton_timeout.IN	:=FALSE;
			eStateTemp	:= eStates;	
			M_Log(eLogType:=ServerityLevelType.INFO,sTextLog:='');
			IF ton_timeout.Q THEN
				RETURN;
			END_IF
		END_IF
		IF ton_timeout.Q THEN	
			ton_timeout.IN	:=FALSE;
			CASE eStates OF	
				E_LoadingStates.ERROR:	
					alarm_temp.Message	:= GenerateErrorMsg(errorType:='M',iState := iStateTemp,errorMsg:='in error state.');
				ELSE
					alarm_temp.Message	:= GenerateErrorMsg(errorType:='M',iState := iStateTemp,errorMsg:='time out');
			END_CASE
//////////////////////////////////////////////////////////states don't want to timeout and trig error//////////////////////////////////////////				
			IF 	eStates<>E_LoadingStates.IDLE AND
				eStates<>E_LoadingStates.WAIT AND 
				eStates<>E_LoadingStates.DETECTION AND
				eStates<>E_LoadingStates.WAIT_READY_TO_TRANSFER AND
				eStates<>E_LoadingStates.WAIT_1	 (*AND 
				(eStates=E_LoadingStates.WAIT_WORKING1_READY_LOAD AND GVL.fb_working1.eState=ePMLState_Execute) AND
				(eStates=E_LoadingStates.WAIT_WORKING2_READY_LOAD AND GVL.fb_working2.eState=ePMLState_Execute)*)
			THEN
				tote_status	:= ToteStatus.MECHANICAL_ERROR;
				isError	:= TRUE; 
				THIS^.pml_adminAlarm.M_SetAlarm(stAdmin:=GVL.PackTags1.Admin,stAlarm:=THIS^.alarm_temp);
				THIS^.pml_adminAlarm.M_SetAlarm(stAdmin:=GVL.PackTags2.Admin,stAlarm:=THIS^.alarm_temp);		
			END_IF
		END_IF
		
		
//////////////////////////////////////////////////////////conditions//////////////////////////////////////////	

		IF GVL.fb_working1.eState=ePMLState_Execute AND GVL.fb_working1.xInbound AND NOT GVL.fb_working1.roller_inbound.photo_sensor[0].Q AND 
			NOT GVL.fb_working1.roller_inbound.photo_sensor[1].Q AND NOT GVL.fb_working1.photo_sensor_tote_detection.Q 
		THEN
			xBeginOutbound_Working1	:= TRUE;
		ELSE
			xBeginOutbound_Working1	:= FALSE;
		END_IF
		IF GVL.fb_working2.eState=ePMLState_Execute AND GVL.fb_working2.xInbound AND NOT GVL.fb_working2.roller_inbound.photo_sensor[0].Q AND 
			NOT GVL.fb_working2.roller_inbound.photo_sensor[1].Q AND NOT GVL.fb_working2.photo_sensor_tote_detection.Q 
		THEN
			xBeginOutbound_Working2	:= TRUE;
		ELSE
			xBeginOutbound_Working2	:= FALSE;
		END_IF
//////////////////////////////////////////////////////////Excute//////////////////////////////////////////
		CASE eStates OF 
				E_LoadingStates.IDLE:	
					ton_timeout.PT	:= T#20MS;				
					eStates	:= E_LoadingStates.INIT;				
				E_LoadingStates.INIT:
					ton_timeout.PT	:= T#5S;
					xOutbound_woking1	:= FALSE;
					xOutbound_woking2	:= FALSE;
					eStates	:= E_LoadingStates.DETECTION;
				E_LoadingStates.DETECTION:
					st_mcAxis.mcMoveAbsolute.Execute	:= FALSE;
					ton_timeout.PT	:= T#5S;
					eTransfer	:= E_Transfer.IDLE;
					//TODO:make sure totestatus is vacant
					IF NOT(roller_assign.photo_sensor[0].Q OR roller_assign.photo_sensor[1].Q OR photo_sensor_diagonal.Q OR
						roller_inbound.photo_sensor[0].Q OR roller_inbound.photo_sensor[1].Q OR photo_sensor_bottom.Q OR
						GVL.fb_working1.roller_preInbound.sensor.Q OR GVL.fb_working2.roller_preInbound.sensor.Q ) 
					THEN				
						eStates	:= E_LoadingStates.WAIT_1;	
					END_IF
					//TODO:make sure totestatus is loaded	
					IF NOT(roller_assign.photo_sensor[0].Q OR roller_assign.photo_sensor[1].Q  OR photo_sensor_bottom.Q OR
						GVL.fb_working1.roller_inbound.photo_sensor[0].Q OR GVL.fb_working2.roller_inbound.photo_sensor[0].Q OR
						GVL.fb_working1.roller_preInbound.sensor.Q OR GVL.fb_working2.roller_preInbound.sensor.Q ) AND 
						roller_inbound.photo_sensor[0].Q AND roller_inbound.photo_sensor[1].Q AND photo_sensor_diagonal.Q
					THEN						
						IF xOutbound_woking1 AND xBeginOutbound_Working1 THEN
							eStates	:= E_LoadingStates.WORKING1_INBOUND_TOTE;
							RETURN;//avoid xOutbound_woking2 works
						END_IF
						IF xOutbound_woking2 AND xBeginOutbound_Working2 THEN

							eStates	:= E_LoadingStates.WORKING2_INBOUND_TOTE;
						END_IF
					END_IF					
					
					
//////////////////////////////////////load/////////////////////////////////			
				E_LoadingStates.WAIT_1:	
					ton_timeout.PT	:= T#100MS;
					IF NOT (roller_assign.photo_sensor[0].Q OR roller_assign.photo_sensor[1].Q OR
						GVL.fb_working1.roller_preInbound.sensor.Q OR GVL.fb_working2.roller_preInbound.sensor.Q) AND ton_timeout.Q
					THEN
						eStates	:= E_LoadingStates.LOAD_UP_POSITION;
					END_IF					
				E_LoadingStates.LOAD_UP_POSITION:	
					ton_timeout.PT	:= T#5S;
					IF NOT (roller_assign.photo_sensor[0].Q OR roller_assign.photo_sensor[1].Q OR
						GVL.fb_working1.roller_preInbound.sensor.Q OR GVL.fb_working2.roller_preInbound.sensor.Q) 
					THEN
						st_mcAxis.mcMoveAbsolute.Execute	:= TRUE;						
						st_mcAxis.rActualPosSet	:= rPos_load;
						st_mcAxis.rVelocitySet	:= 300;
						IF st_mcAxis.mcMoveAbsolute.Done THEN
							st_mcAxis.mcMoveAbsolute.Execute	:= FALSE;
							eTransfer	:= E_Transfer.LOAD;
							eStates	:= E_LoadingStates.WAIT_READY_TO_TRANSFER;
						END_IF
					END_IF
			
				E_LoadingStates.WAIT_READY_TO_TRANSFER:
					ton_timeout.PT	:= T#30S;
					IF ton_timeout.Q THEN
						tote_status	:= ToteStatus.TIMEOUT_WAITING_FOR_NEW_TOTE;
						////////abort inbound command if woking is in awaiting new tote////////////////
//						subData.Topic	:= E_Topics.WORKING1_ABORT_INBOUND;
//						GVL.PubSubService.Publish(topic:=E_Topics.WORKING1_ABORT_INBOUND,data:= subData);
//						subData.Topic	:= E_Topics.WORKING2_ABORT_INBOUND;
//						GVL.PubSubService.Publish(topic:=E_Topics.WORKING2_ABORT_INBOUND,data:= subData);							
					ELSE
						tote_status	:= ToteStatus.AWAITING_INBOUND_AVAILABILITY;
					END_IF
					logtech_load_command	:= LogTechControlCmd.READY_TO_RECEIVE;
					IF photo_sensor_bottom.Q THEN//todo:remove while onsite
						logtech_load_status	:= LogTechTransferStatus.READY_TO_TRANSFER;
					END_IF
					IF logtech_load_status=LogTechTransferStatus.READY_TO_TRANSFER THEN
						logtech_load_status	:= LogTechTransferStatus.UNKNOWN;//todo:remove this while on site
						eStates	:= E_LoadingStates.ROLLER_Y_LOAD;
					END_IF									
				E_LoadingStates.ROLLER_Y_LOAD:
					ton_timeout.PT	:= T#3S;
					tote_status	:= ToteStatus.INBOUNDING;
					logtech_load_command	:= LogTechControlCmd.RECEIVING_TOTE;
					roller_inbound.roller.forward	:= TRUE;
					roller_inbound_assist.roller.forward	:= TRUE;
					IF roller_inbound.photo_sensor[0].Q AND roller_inbound.photo_sensor[1].Q AND photo_sensor_diagonal.Q AND NOT photo_sensor_bottom.Q THEN
						roller_inbound.roller.forward	:= FALSE;
						roller_inbound_assist.roller.forward	:= FALSE;
						eStates	:= E_LoadingStates.WAIT;
					END_IF
				E_LoadingStates.WAIT:
					ton_timeout.PT	:= T#500MS;
					roller_inbound.roller.forward	:= TRUE;
					roller_inbound_assist.roller.forward	:= TRUE;					
					IF ton_timeout.Q THEN
						roller_inbound.roller.forward	:= FALSE;
						roller_inbound_assist.roller.forward	:= FALSE;						
						eStates	:= E_LoadingStates.LOAD_DOWN_POSITION;
						logtech_load_command	:= LogTechControlCmd.RECEIVE_TOTE_FINISHED;
					END_IF				
				E_LoadingStates.LOAD_DOWN_POSITION:
					ton_timeout.PT	:= T#5S;
					st_mcAxis.mcMoveAbsolute.Execute	:= TRUE;						
					st_mcAxis.rActualPosSet	:= rPos_unload;
					st_mcAxis.rVelocitySet	:= 300;
					IF st_mcAxis.mcMoveAbsolute.Done THEN
						st_mcAxis.mcMoveAbsolute.Execute	:= FALSE;
						tote_status	:= ToteStatus.LOADED;
						eStates	:= E_LoadingStates.DETECTION;
					END_IF							
					
					
					
		///////////////////////////////unload to working1/////////////////////////////////	
					
				E_LoadingStates.WORKING1_INBOUND_TOTE:	
					IF xOutbound_woking1 THEN	
						tote_status	:= ToteStatus.AWAITING_OUTBOUND_AVAILABILITY;
						eStates	:= E_LoadingStates.WAIT_WORKING1_READY_LOAD;
						subData.Topic	:= E_Topics.WORKING1_BEGIN_INBOUND;
						GVL.PubSubService.Publish(topic:=E_Topics.WORKING1_BEGIN_INBOUND,data:= subData);	
					ELSE
						ton_timeout.IN	:= FALSE;
					END_IF				
				E_LoadingStates.WAIT_WORKING1_READY_LOAD:
					IF xOutbound_woking1 THEN
						ton_timeout.PT	:= T#3S;//should be shorter than woriking's inbound process
						IF valve_left_door.retracted AND GVL.fb_working1.eState=ePMLState_Execute THEN
							tote_status	:= ToteStatus.OUTBOUNDING;
							eStates	:= E_LoadingStates.ROLLER_UNLOAD_WORKING1;
						END_IF	
					ELSE
						ton_timeout.IN	:= FALSE;	
					END_IF		
				E_LoadingStates.ROLLER_UNLOAD_WORKING1:
					IF xOutbound_woking1 THEN
						tote_status	:= ToteStatus.OUTBOUNDING;
						roller_assign.roller.forward	:= TRUE;
						IF NOT photo_sensor_diagonal.Q THEN
							eStates	:= E_LoadingStates.WAIT_FINISH_OUTBOUND1;
						END_IF	
					ELSE
						ton_timeout.IN	:= FALSE;
					END_IF			
				E_LoadingStates.WAIT_FINISH_OUTBOUND1:
					IF xOutbound_woking1 THEN
						tote_status	:= ToteStatus.OUTBOUNDING;
						roller_assign.roller.forward	:= TRUE;
						IF NOT roller_assign.photo_sensor[0].Q THEN
							roller_assign.roller.forward	:= FALSE;
							tote_status	:= ToteStatus.VACANT;
							xOutbound_woking1	:= FALSE;
							xBeginOutbound_Working1	:= FALSE;						
							eStates	:= E_LoadingStates.DONE;
						END_IF	
					ELSE
						ton_timeout.IN	:= FALSE;
					END_IF				



		///////////////////////////////unload to working2/////////////////////////////////
						
				E_LoadingStates.WORKING2_INBOUND_TOTE:	
					IF xOutbound_woking2 THEN	
						tote_status	:= ToteStatus.AWAITING_OUTBOUND_AVAILABILITY;
						subData.Topic	:= E_Topics.WORKING2_BEGIN_INBOUND;
						GVL.PubSubService.Publish(topic:=E_Topics.WORKING2_BEGIN_INBOUND,data:= subData);				
						eStates	:= E_LoadingStates.WAIT_WORKING2_READY_LOAD;	
					ELSE
						ton_timeout.IN	:= FALSE;
					END_IF
				E_LoadingStates.WAIT_WORKING2_READY_LOAD:
					IF xOutbound_woking2 THEN	
						ton_timeout.PT	:= T#3S;//should be shorter than woriking's inbound process
						IF valve_right_door.retracted AND GVL.fb_working2.eState=ePMLState_Execute THEN
							tote_status	:= ToteStatus.OUTBOUNDING;
							eStates	:= E_LoadingStates.ROLLER_UNLOAD_WORKING2;
						END_IF	
					ELSE
						ton_timeout.IN	:= FALSE;
					END_IF			
				E_LoadingStates.ROLLER_UNLOAD_WORKING2:
					IF xOutbound_woking2 THEN	
						tote_status	:= ToteStatus.OUTBOUNDING;
						roller_assign.roller.backward	:= TRUE;
						IF NOT photo_sensor_diagonal.Q THEN
							eStates	:= E_LoadingStates.WAIT_FINISH_OUTBOUND2;
						END_IF	
					ELSE
						ton_timeout.IN	:= FALSE;	
					END_IF		
				E_LoadingStates.WAIT_FINISH_OUTBOUND2:
					IF xOutbound_woking2 THEN
						tote_status	:= ToteStatus.OUTBOUNDING;	
						roller_assign.roller.backward	:= TRUE;
						IF NOT roller_assign.photo_sensor[1].Q THEN
							roller_assign.roller.backward	:= FALSE;
							tote_status	:= ToteStatus.VACANT;
							xOutbound_woking2	:= FALSE;
							xBeginOutbound_Working2	:= FALSE;						
							eStates	:= E_LoadingStates.DONE;
						END_IF	
					ELSE
						ton_timeout.IN	:= FALSE;	
					END_IF	

				E_LoadingStates.DONE:
					eStates	:= E_LoadingStates.DETECTION;	
		END_CASE


	
		
	ePMLProtUnitMode_Maintenance, ePMLUnitMode_Service:	
		;			
	ePMLProtUnitMode_Manual:		//Manaul

END_CASE
END_METHOD

{attribute 'object_name' := 'M_Holding'}
METHOD M_Holding
CASE fbUnitModeManager.eModeStatus OF
	ePMLProtUnitMode_Production:		//Mode Production
		//Finisch the actual seperationstep	

	ePMLProtUnitMode_Maintenance:
		M_StateComplete();
END_CASE
END_METHOD

{attribute 'object_name' := 'M_Idle'}
METHOD M_Idle
ftrig_agingTest(CLK	:= bAging_test);
IF 	ftrig_agingTest.Q THEN
	iAging_test	:= 10;
END_IF
IF bAging_test THEN
	IF iAging_test=0 THEN
		iAging_test	:= 1;
	END_IF	
END_IF
M_agingTest(1.0);
END_METHOD

//RISK:it is a risk for people to make the lift door move down automatically
//todo:use case to reprogrma to easy debug the program?
METHOD M_LockRequest_1 : BOOL
VAR_INPUT

END_VAR
VAR
	
END_VAR
(*
left gate lock request	right gate is unlocked but closed	no tote between loading AND working2 	left door up AND right door down	left gate lock
						right gate locked															left door up						left gate lock
*)
M_LockRequest_1	:= FALSE;

xLocking1	:= TRUE;
IF MAIN.safety_2.safety_door_array[0]=SafetyDoorStatus.LOCKED THEN//right gate locked
	//left door up
	valve_left_door.extend	:= FALSE;
	valve_left_door.retract	:= TRUE;
	IF NOT valve_left_door.extended AND valve_left_door.retracted THEN
		xLocking1	:= FALSE;
		M_LockRequest_1	:= TRUE;
	END_IF	
//	ELSIF MAIN.safety_2.door_closed THEN//right gate unlocked but closed
ELSIF MAIN.safety_2.lift_door_right.Q THEN//right gate unlocked but lift right door is down
	IF  NOT (roller_assign.photo_sensor[1].Q OR GVL.fb_working2.roller_inbound.photo_sensor[0].Q) THEN//no tote between loading AND working2
		//left door up AND right door down
		valve_left_door.extend		:= FALSE;
		valve_left_door.retract		:= TRUE;
		valve_right_door.extend		:= TRUE;
		valve_right_door.retract	:= FALSE;		
		IF NOT valve_left_door.extended AND valve_left_door.retracted AND valve_right_door.extended AND NOT valve_right_door.retracted THEN
			xLocking1	:= FALSE;
			M_LockRequest_1	:= TRUE;
		END_IF		
	END_IF 
END_IF
END_METHOD

//RISK:it is a risk for people to make the lift door move down automatically
//todo:use case to reprogrma to easy debug the program?
METHOD M_LockRequest_2 : BOOL
VAR
	
END_VAR
(*
right gate lock request		left gate is unlocked but closed	no tote between loading and working1	left door down and right door up	right gate lock
							left gate locked															right door up						right gate lock
*)
M_LockRequest_2	:= FALSE;	
xLocking2	:= TRUE;
IF MAIN.safety_1.safety_door_array[0]=SafetyDoorStatus.LOCKED THEN//left gate locked
	//right door up
	valve_right_door.extend		:= FALSE;
	valve_right_door.retract	:= TRUE;
	IF NOT valve_right_door.extended AND valve_right_door.retracted THEN
		xLocking2	:= FALSE;
		M_LockRequest_2	:= TRUE;
	END_IF	
//	ELSIF MAIN.safety_1.door_closed THEN//left gate unlocked but closed
ELSIF MAIN.safety_1.lift_door_left.Q THEN//right gate unlocked but lift left door is down
	IF NOT (roller_assign.photo_sensor[0].Q OR GVL.fb_working1.roller_inbound.photo_sensor[0].Q) THEN//no tote between loading AND working1
		//right door up AND left door down
		valve_left_door.extend		:= TRUE;
		valve_left_door.retract		:= FALSE;
		valve_right_door.extend		:= FALSE;
		valve_right_door.retract	:= TRUE	;		
		IF valve_left_door.extended AND NOT valve_left_door.retracted AND NOT valve_right_door.extended AND valve_right_door.retracted THEN
			xLocking2	:= FALSE;
			M_LockRequest_2	:= TRUE;
		END_IF		
	END_IF 
END_IF
END_METHOD

METHOD M_mapping : BOOL
VAR_INPUT
END_VAR
/////////////////////////////////////digital input////////////////////////////////////////

roller_assign.roller.err(D:= G_IO.arDI[2].Ch[0],on_ms:=3000,off_ms:=80);	
roller_assign.photo_sensor[0](D:= arIOLinkTx_Lift[7].InputByte[1].2,on_ms:=100,off_ms:=100);
roller_assign.photo_sensor[1](D:=  arIOLinkTx_Lift[7].InputByte[0].2 ,on_ms:=100,off_ms:=100);

roller_inbound.roller.err(D:= G_IO.arDI[2].Ch[1],on_ms:=3000,off_ms:=80);	
roller_inbound.photo_sensor[0](D:= arIOLinkTx_Lift[7].InputByte[1].0,on_ms:=100,off_ms:=100);   //料筐检测0(到位)
roller_inbound.photo_sensor[1](D:= arIOLinkTx_Lift[7].InputByte[0].0,on_ms:=100,off_ms:=100);  //料筐检测1(到位)

roller_inbound_assist.roller.err(D:= G_IO.arDI[2].Ch[2],on_ms:=3000,off_ms:=80);
EDM_KM            							:= G_IO.arDI[2].Ch[3];       //P24_sto          

photo_sensor_diagonal(D:= arIOLinkTx_Lift[7].InputByte[1].1,on_ms:=100,off_ms:=100);  //料筐检测2(对角)
photo_sensor_bottom(D:= arIOLinkTx_Lift[7].InputByte[0].1,on_ms:=100,off_ms:=100);    //todo:modify while onsite

valve_left_door.retracted			:= arIOLinkQualifier_Lift.CH[0].1 ;
valve_left_door.extended			:= arIOLinkQualifier_Lift.CH[1].1 ;
valve_right_door.retracted			:= arIOLinkQualifier_Lift.CH[2].1 ;
valve_right_door.extended			:= arIOLinkQualifier_Lift.CH[3].1 ;

st_mcAxis.limit_sensor_positive		:= arIOLinkQualifier_Lift.CH[4].0;
st_mcAxis.limit_sensor_negative		:= arIOLinkQualifier_Lift.CH[4].1;
st_mcAxis.limit_sensor_home			:= arIOLinkQualifier_Lift.CH[5].1;


/////////////////////////////////////digital output////////////////////////////////////////
G_IO.arDO[2].Ch[0]	:= roller_assign.roller.forward;
G_IO.arDO[2].Ch[1]	:= roller_assign.roller.backward;
G_IO.arDO[2].Ch[2]	:= roller_inbound.roller.forward;
G_IO.arDO[2].Ch[3]	:= roller_inbound.roller.backward;
G_IO.arDO[2].Ch[4]	:= roller_inbound_assist.roller.forward;
G_IO.arDO[2].Ch[5]	:= roller_inbound_assist.roller.backward;

G_IO.arDO[6].Ch[3] :=valve_left_door.retract;
G_IO.arDO[6].Ch[2] :=valve_left_door.extend;
G_IO.arDO[7].Ch[3] :=valve_right_door.retract;
G_IO.arDO[7].Ch[2] :=valve_right_door.extend;


G_IO.arDO[2].Ch[14] := floodlight;  //照明灯

/////////////////////////////////////axis config////////////////////////////////////////
mcAxis
(
	ZSP		:=  (st_mcAxis.limit_sensor_positive OR st_mcAxis.xHoming) AND 
				(NOT (roller_assign.photo_sensor[0].Q OR roller_assign.photo_sensor[1].Q OR
				GVL.fb_working1.roller_preInbound.sensor.Q OR GVL.fb_working2.roller_preInbound.sensor.Q) OR eState<>ePMLState_Execute), //TODO link to digital input
	
	ZSN		:=  (st_mcAxis.limit_sensor_negative OR st_mcAxis.xHoming) AND 
				(NOT (roller_assign.photo_sensor[0].Q OR roller_assign.photo_sensor[1].Q OR
				GVL.fb_working1.roller_preInbound.sensor.Q OR GVL.fb_working2.roller_preInbound.sensor.Q) OR eState<>ePMLState_Execute), //TODO link to digital input
	IN_OUT	:= st_mcAxis	, 
	AXIS	:= AxisRef	, 
);
st_mcAxis.bPosSensorShow	:= TRUE;
st_mcAxis.bNegSensorShow	:= TRUE;
st_mcAxis.bStopButtonShow	:= TRUE;
st_mcAxis.rMaxAcceleration	:= 50000;
st_mcAxis.rMaxDeceleration	:= 50000;
st_mcAxis.rMaxJerk			:= 500000;
st_mcAxis.rAcceleration	:= 2500;
st_mcAxis.rDeceleration	:= 2500;
st_mcAxis.rJerk			:= 12500;
st_mcAxis.rMaxVelocity		:= 100;
st_mcAxis.rMaxDistance		:= 50;
st_mcAxis.bPosSen	:=  st_mcAxis.limit_sensor_positive AND 
						(NOT (roller_assign.photo_sensor[0].Q OR roller_assign.photo_sensor[1].Q OR
						GVL.fb_working1.roller_inbound.photo_sensor[0].Q OR GVL.fb_working2.roller_inbound.photo_sensor[0].Q) OR eState<>ePMLState_Execute);

st_mcAxis.bNegSen	:=  st_mcAxis.limit_sensor_negative AND 
						(NOT (roller_assign.photo_sensor[0].Q OR roller_assign.photo_sensor[1].Q OR
						GVL.fb_working1.roller_inbound.photo_sensor[0].Q OR GVL.fb_working2.roller_inbound.photo_sensor[0].Q) OR eState<>ePMLState_Execute);

st_mcAxis.mcHome.bCalibrationCam	:= st_mcAxis.limit_sensor_home;
st_mcAxis.bPositionSensor	:= st_mcAxis.limit_sensor_home;
st_mcAxis.bdirFW	:= TRUE;
st_mcAxis.sNetID := '192.168.17.27.5.1';
st_mcAxis.nSlaveAddr	:= 1011;
st_mcAxis.rToqueLimitSet	:= 120;

/////////////////////////////////////LogTech/////////////////////////////////////////////
END_METHOD

METHOD M_Reset
VAR_INPUT
END_VAR
//Take away all commands
IF GVL.stChangeIntoProduction.bYesReset THEN
;
END_IF
END_METHOD

{attribute 'object_name' := 'M_Resetting'}
METHOD M_Resetting
CASE fbUnitModeManager.eModeStatus OF
	ePMLProtUnitMode_Production:		//Production, Mantainance, Manual
		st_mcAxis.mcStop.Execute	:= FALSE;
		st_mcAxis.mcReset.Execute	:= TRUE;
		eTransfer	:= E_Transfer.IDLE;	
		ton_timeout.IN	:= FALSE;
		M_StateComplete();
	
	ePMLProtUnitMode_Maintenance, ePMLProtUnitMode_Manual, ePMLUnitMode_Service:
		M_StateComplete();
END_CASE
END_METHOD

{attribute 'object_name' := 'M_Starting'}
METHOD M_Starting
CASE fbUnitModeManager.eModeStatus OF
	ePMLProtUnitMode_Production:		//Production, Mantainance, Manual
		st_mcAxis.mcPower.Enable	:= TRUE;
		IF 	photo_sensor_diagonal.Q AND 
			roller_inbound.photo_sensor[0].Q AND
			roller_inbound.photo_sensor[1].Q AND
			NOT(roller_assign.photo_sensor[0].Q OR roller_assign.photo_sensor[1].Q) AND
			NOT photo_sensor_bottom.Q AND
			ABS(AxisRef.NcToPlc.ActPos-rPos_unload)<1
		THEN
			tote_status	:= ToteStatus.LOADED;
			eStates	:= E_LoadingStates.IDLE;
		END_IF
		IF NOT(roller_assign.photo_sensor[0].Q OR roller_assign.photo_sensor[1].Q OR photo_sensor_diagonal.Q
		OR roller_inbound.photo_sensor[0].Q OR roller_inbound.photo_sensor[1].Q OR photo_sensor_bottom.Q) THEN
			tote_status	:= ToteStatus.VACANT;
			eStates	:= E_LoadingStates.IDLE;
		END_IF		
		IF st_mcAxis.mcPower.Status THEN
			M_StateComplete();
		END_IF
		
	ePMLProtUnitMode_Maintenance, ePMLProtUnitMode_Manual, ePMLUnitMode_Service:
		M_StateComplete();
END_CASE
END_METHOD

{attribute 'object_name' := 'M_Stopping'}
METHOD M_Stopping
CASE fbUnitModeManager.eModeStatus OF
	ePMLProtUnitMode_Production, ePMLProtUnitMode_Manual:
//////////////////////////////////////////////////////////timeout//////////////////////////////////////////	
		ton_timeout.IN	:= TRUE;
		ton_timeout.PT := T#2S;
		IF ton_timeout.Q THEN
			ton_timeout.IN	:= FALSE;
			M_StateComplete();
		END_IF
	ePMLProtUnitMode_Maintenance, ePMLUnitMode_Service:
		M_StateComplete();	
			//not defined
END_CASE
END_METHOD

{attribute 'object_name' := 'M_Undefined'}
METHOD M_Undefined

bUndefinedDone					:= TRUE;
END_METHOD

METHOD M_UnlockRequest : BOOL
VAR_INPUT
	sInstanceName	: STRING;
END_VAR
VAR
	
END_VAR
(*
left gate unlock request	working1 stopped	no tote between loading AND working1	left door down		left gate unlock
												tote between loading AND working1		left door up		left gate unlock				
*)
IF sInstanceName='safety_1' THEN
	xUnlocking1	:= TRUE;
	IF GVL.fb_working1.eState<>ePMLState_Stopping AND GVL.fb_working1.eState<>ePMLState_Execute THEN//working1 stopped
		IF GVL.fb_working1.roller_inbound.photo_sensor[0].Q OR roller_assign.photo_sensor[0].Q THEN//tote between loading AND working1
			//left door up
			valve_left_door.extend	:= FALSE;
			valve_left_door.retract	:= TRUE;
			IF NOT valve_left_door.extended AND valve_left_door.retracted THEN
				xUnlocking1	:= FALSE;
				M_unlockRequest	:= TRUE;
			END_IF	
		ELSE//no tote between loading AND working1
			//left door down
			valve_left_door.extend	:= TRUE;
			valve_left_door.retract	:= FALSE;
			IF valve_left_door.extended AND NOT valve_left_door.retracted AND MAIN.safety_1.lift_door_left.Q THEN
				xUnlocking1	:= FALSE;
				M_unlockRequest	:= TRUE;
			END_IF
		END_IF
	END_IF
END_IF
(*
right gate unlock request	working2 stopped	no tote between loading and working2 	right door down		right gate unlock
												tote between loading and working2 		right door up		right gate unlock
*)
IF sInstanceName='safety_2' THEN
	xUnlocking2	:= TRUE;
	IF GVL.fb_working2.eState<>ePMLState_Stopping AND GVL.fb_working2.eState<>ePMLState_Execute THEN//working2 stopped
		IF GVL.fb_working2.roller_inbound.photo_sensor[0].Q OR roller_assign.photo_sensor[1].Q THEN//tote between loading AND working2
			//right door up
			valve_right_door.extend		:= FALSE;
			valve_right_door.retract	:= TRUE;
			IF NOT valve_right_door.extended AND valve_right_door.retracted THEN
				xUnlocking2	:= FALSE;
				M_unlockRequest	:= TRUE;
			END_IF	
		ELSE//no tote between loading AND working2
			//right door down
			valve_right_door.extend		:= TRUE;
			valve_right_door.retract	:= FALSE;
			IF valve_right_door.extended AND NOT valve_right_door.retracted AND MAIN.safety_1.lift_door_right.Q THEN
				xUnlocking2	:= FALSE;
				M_unlockRequest	:= TRUE;
			END_IF
		END_IF
	END_IF
END_IF
END_METHOD

METHOD ParseStateToString : STRING
VAR_INPUT
END_VAR
CASE THIS^.eStates OF
	E_LoadingStates.IDLE:		
		ParseStateToString	:= 'IDLE';
	E_LoadingStates.INIT:
		ParseStateToString	:= 'INIT';
	E_LoadingStates.CHECK:
		ParseStateToString	:= 'CHECK';
	E_LoadingStates.WAIT:
		ParseStateToString	:= 'WAIT';
	E_LoadingStates.WAIT_1:
		ParseStateToString	:= 'WAIT_1';
	E_LoadingStates.DETECTION:
		ParseStateToString	:= 'DETECTION';
	E_LoadingStates.LOADING:
		ParseStateToString	:= 'LOADING';
	E_LoadingStates.UNLOADING:
		ParseStateToString	:= 'UNLOADING';
	E_LoadingStates.WAIT_WORKING1_READY_LOAD:
		ParseStateToString	:= 'WAIT_WORKING1_READY_LOAD';
	E_LoadingStates.WAIT_WORKING2_READY_LOAD:
		ParseStateToString	:= 'WAIT_WORKING2_READY_LOAD';
	E_LoadingStates.LIFT_POSITION_LOAD:
		ParseStateToString	:= 'LIFT_POSITION_LOAD';
	E_LoadingStates.LIFT_POSITION_UNLOAD:
		ParseStateToString	:= 'LIFT_POSITION_UNLOAD';
	E_LoadingStates.LIFT_UP:
		ParseStateToString	:= 'LIFT_UP';
	E_LoadingStates.ROLLER_LOAD:
		ParseStateToString	:= 'ROLLER_LOAD';
	E_LoadingStates.ROLLER_UNLOAD_WORKING1:
		ParseStateToString	:= 'ROLLER_UNLOAD_WORKING1';
	E_LoadingStates.ROLLER_UNLOAD_WORKING2:
		ParseStateToString	:= 'ROLLER_UNLOAD_WORKING2';		
	E_LoadingStates.WAIT_FINISH_OUTBOUND1:		
		ParseStateToString	:= 'WAIT_FINISH_OUTBOUND1';
	E_LoadingStates.WAIT_FINISH_OUTBOUND2:		
		ParseStateToString	:= 'WAIT_FINISH_OUTBOUND2';
	E_LoadingStates.AGING_STATE_0:		
		ParseStateToString	:= 'AGING_STATE_0';
	E_LoadingStates.AGING_STATE_1:		
		ParseStateToString	:= 'AGING_STATE_1';
	E_LoadingStates.WAIT_READY_TO_TRANSFER:		
		ParseStateToString	:= 'WAIT_READY_TO_TRANSFER';
	E_LoadingStates.LOAD_UP_POSITION:		
		ParseStateToString	:= 'LOAD_UP_POSITION';
	E_LoadingStates.LOAD_DOWN_POSITION:		
		ParseStateToString	:= 'LOAD_DOWN_POSITION';
	E_LoadingStates.ROLLER_Y_LOAD:		
		ParseStateToString	:= 'ROLLER_Y_LOAD';
	E_LoadingStates.WORKING1_INBOUND_TOTE:		
		ParseStateToString	:= 'WORKING1_INBOUND_TOTE';	
	E_LoadingStates.WORKING2_INBOUND_TOTE:
		ParseStateToString	:= 'WORKING2_INBOUND_TOTE';
	E_LoadingStates.DONE:
		ParseStateToString	:= 'DONE';
	E_LoadingStates.ERROR:
		ParseStateToString	:= 'ERROR';
ELSE
		ParseStateToString	:= 'UNKNOW STATE';
END_CASE
END_METHOD

END_FUNCTION_BLOCK

// ---- Mian/FB_autoStore.TcPOU
FUNCTION_BLOCK FB_autoStore EXTENDS FB_Generic
VAR_INPUT
END_VAR
VAR_OUTPUT
END_VAR
VAR
	lamp			: BOOL;	
	eStates			: E_AutoStore_States := E_AutoStore_States.IDLE;;
	eStateTemp		: E_AutoStore_States := E_AutoStore_States.IDLE;
	
	mcAxis_lift 			: FB_MotionAxis_MC;
	st_mcAxis_lift 			: ST_MotionAxis_MC;
	AxisRef_lift			: AXIS_REF;
	
	mcAxis_transfer 		: FB_MotionAxis_MC;
	st_mcAxis_transfer		: ST_MotionAxis_MC;
	AxisRef_transfer		: AXIS_REF;
	
	door_closed						: BOOL;
	button_start					: BOOL;	
	button_stop						: BOOL;	
	sensor_lift_atDownPos			: BOOL;
	sensor_transfer_atWorkingPos	: BOOL;
	sensor_transfer_atFeedingPos	: BOOL;
	
	bUpStairs						: BOOL;
	bExchangeTote					: BOOL;
	
	
	autostore_status	: AutostoreStatus;
END_VAR	
VAR PERSISTENT
	rPos_lift_up				: REAL;//340
	rPos_lift_down				: REAL;
	rPos_transfer_feeding		: REAL;
	rPos_transfer_working		: REAL;//636	
END_VAR

SUPER^();
IF sInstanceName='autoStore_1' THEN
	rPos_lift_up				:= 350;
	rPos_lift_down				:= 0;
	rPos_transfer_feeding		:= 0;
	rPos_transfer_working		:= 656;	
END_IF
IF sInstanceName='autoStore_2' THEN
	rPos_lift_up				:= 350;
	rPos_lift_down				:= 0;
	rPos_transfer_feeding		:= 0;
	rPos_transfer_working		:= 624;	
END_IF
IF sInstanceName='autoStore_1' THEN
	IF NOT subscribed THEN
		GVL.PubSubService.Subscribe(E_Topics.AUTOSTORE1_EXCHANGE,sInstanceName,THIS^);
		subscribed	:= TRUE;
	END_IF
END_IF
IF sInstanceName='autoStore_2' THEN
	IF NOT subscribed THEN
		GVL.PubSubService.Subscribe(E_Topics.AUTOSTORE2_EXCHANGE,sInstanceName,THIS^);
		subscribed	:= TRUE;
	END_IF
END_IF

//sComponent_name		:= _sInstanceName;
//iComponetID			:= ModuleID.SAMPLE1;

infoLevel	:= ServerityLevelType.WARNING;

(*
Description: 
the callback that will be invoked when there is a publish for what the subscriber was subscribed to.
*)
METHOD Callback
VAR_INPUT
	data : PubSubData;
END_VAR
IF door_closed THEN
	IF sInstanceName='autoStore_1' THEN
		CASE data.Topic OF
			E_Topics.AUTOSTORE1_EXCHANGE:
				IF autostore_status<>AutostoreStatus.EXCHANGING THEN
					bExchangeTote	:= TRUE;	
				END_IF
		END_CASE	
	END_IF
	IF sInstanceName='autoStore_2' THEN
		CASE data.Topic OF
			E_Topics.AUTOSTORE2_EXCHANGE:
				IF autostore_status<>AutostoreStatus.EXCHANGING THEN
					bExchangeTote	:= TRUE;	
				END_IF		
		END_CASE	
	END_IF
END_IF
END_METHOD

{attribute 'object_name' := 'M_Aborting'}
METHOD M_Aborting
CASE fbUnitModeManager.eModeStatus OF	
	ePMLProtUnitMode_Production, ePMLProtUnitMode_Manual:		

		st_mcAxis_lift.mcMoveAbsolute.Execute		:= FALSE;
		st_mcAxis_lift.mcStop.Execute				:= TRUE;	
		st_mcAxis_transfer.mcMoveAbsolute.Execute	:= FALSE;
		st_mcAxis_transfer.mcStop.Execute			:= TRUE;
		iAging_test	:= 0;
		M_StateComplete();
			
	ePMLProtUnitMode_Maintenance, ePMLUnitMode_Service:
		
		M_StateComplete();
END_CASE
END_METHOD

METHOD M_agingTest : BOOL
VAR_INPUT
	rVelocity_percent	: REAL;
END_VAR
END_METHOD

{attribute 'object_name' := 'M_Completing'}
METHOD M_Completing
CASE fbUnitModeManager.eModeStatus OF
	ePMLProtUnitMode_Production:
		;
END_CASE
END_METHOD

{attribute 'object_name' := 'M_Execute'}
METHOD M_Execute
IF door_closed THEN
	st_mcAxis_transfer.mcStop.Execute	:= FALSE;
	st_mcAxis_lift.mcStop.Execute		:= FALSE;
	st_mcAxis_transfer.mcReset.Execute	:= TRUE;
	st_mcAxis_lift.mcReset.Execute		:= TRUE;	
ELSE
	st_mcAxis_transfer.mcStop.Execute	:= TRUE;
	st_mcAxis_lift.mcStop.Execute		:= TRUE;
	RETURN;
END_IF
CASE fbUnitModeManager.eModeStatus OF
	ePMLProtUnitMode_Production:		//Mode Production
//////////////////////////////////////////////////////////timeout//////////////////////////////////////////	
		iStateTemp	:= eStateTemp;
		ton_timeout();
		IF eStateTemp=eStates THEN
			ton_timeout.IN	:=TRUE;
		ELSE
			ton_timeout.IN	:=FALSE;
			eStateTemp	:= eStates;	
			M_Log(eLogType:=ServerityLevelType.INFO,sTextLog:='');
			IF ton_timeout.Q THEN
				RETURN;
			END_IF
		END_IF
		IF ton_timeout.Q THEN	
			ton_timeout.IN	:=FALSE;
			CASE eStates OF	
				E_AutoStore_States.ERROR:	
					alarm_temp.Message	:= GenerateErrorMsg(errorType:='M',iState := iStateTemp,errorMsg:='in error state.');
				ELSE
				alarm_temp.Message	:= GenerateErrorMsg(errorType:='M',iState := iStateTemp,errorMsg:='time out');
			END_CASE
//////////////////////////////////////////////////////////states don't want to timeout and trig error//////////////////////////////////////////				
			IF 	eStates<>E_AutoStore_States.IDLE AND
				eStates<>E_AutoStore_States.WAIT AND
				eStates<>E_AutoStore_States.WAIT_CMD
			THEN 
				IF sInstanceName='autoStore_1' THEN
					GVL.pml_adminAlarm.M_SetAlarm(stAdmin:=GVL.PackTags1.Admin,stAlarm:=alarm_temp);
				END_IF
				IF sInstanceName='autoStore_2' THEN
					GVL.pml_adminAlarm.M_SetAlarm(stAdmin:=GVL.PackTags2.Admin,stAlarm:=alarm_temp);
				END_IF					
			END_IF
		END_IF
//////////////////////////////////////////////////////////auto running process//////////////////////////////////////////			
		CASE eStates OF 
				E_AutoStore_States.IDLE:
					ton_timeout.PT	:= T#1MS;						
					eStates	:= E_AutoStore_States.INIT;				
				E_AutoStore_States.INIT:
					ton_timeout.PT	:= T#1S;
					st_mcAxis_transfer.mcMoveAbsolute.Execute	:= FALSE;
					st_mcAxis_lift.mcMoveAbsolute.Execute	:= FALSE;
					autostore_status	:= AutostoreStatus.UNKNOWN;
					eStates	:= E_AutoStore_States.WAIT; 
				E_AutoStore_States.WAIT:
					ton_timeout.PT	:= T#10S;
					eStates	:= E_AutoStore_States.WAIT_CMD; 
				E_AutoStore_States.WAIT_CMD:
					IF bExchangeTote OR button_start THEN
						bExchangeTote	:= FALSE;
						autostore_status	:= AutostoreStatus.EXCHANGING;
						eStates	:= E_AutoStore_States.LIFT_MOVE_DOWN;
					END_IF
				////////////////////////////lift move down///////////////////////////////////		
				E_AutoStore_States.LIFT_MOVE_DOWN:	
					st_mcAxis_lift.mcMoveAbsolute.Execute	:= TRUE;					
					st_mcAxis_lift.rActualPosSet	:= rPos_lift_down;
					st_mcAxis_lift.rVelocitySet		:= 400;					
					IF st_mcAxis_lift.mcMoveAbsolute.Done THEN
						st_mcAxis_lift.mcMoveAbsolute.Execute	:= FALSE;
						eStates	:= E_AutoStore_States.LIFT_DOWN_SENSOR_DETECTED;
					END_IF
				E_AutoStore_States.LIFT_DOWN_SENSOR_DETECTED:	
					IF TRUE OR sensor_lift_atDownPos THEN
						IF bUpStairs THEN
							eStates	:= E_AutoStore_States.TRANSFER_MOVE_FEEDING;
							bUpStairs	:= FALSE;
						ELSE
							eStates	:= E_AutoStore_States.TRANSFER_MOVE_WORKING;
							bUpStairs	:= TRUE;
						END_IF					
					END_IF
				////////////////////////////upstairs///////////////////////////////////	
				E_AutoStore_States.TRANSFER_MOVE_FEEDING:	
					st_mcAxis_transfer.mcMoveAbsolute.Execute	:= TRUE;					
					st_mcAxis_transfer.rActualPosSet	:= rPos_transfer_feeding;
					st_mcAxis_transfer.rVelocitySet		:= 600;					
					IF st_mcAxis_transfer.mcMoveAbsolute.Done THEN
						st_mcAxis_transfer.mcMoveAbsolute.Execute	:= FALSE;
						eStates	:= E_AutoStore_States.TRANSFER_FEEDING_SENSOR_DETECTED;
					END_IF				

				E_AutoStore_States.TRANSFER_FEEDING_SENSOR_DETECTED:
					IF sensor_transfer_atFeedingPos OR TRUE THEN//todo:add this sensor
						eStates	:= E_AutoStore_States.LIFT_MOVE_UP;
					END_IF									
				////////////////////////////downstairs///////////////////////////////////		
				E_AutoStore_States.TRANSFER_MOVE_WORKING:	
					st_mcAxis_transfer.mcMoveAbsolute.Execute	:= TRUE;					
					st_mcAxis_transfer.rActualPosSet	:= rPos_transfer_working;
					st_mcAxis_transfer.rVelocitySet		:= 600;					
					IF st_mcAxis_transfer.mcMoveAbsolute.Done THEN
						st_mcAxis_transfer.mcMoveAbsolute.Execute	:= FALSE;
						eStates	:= E_AutoStore_States.TRANSFER_WORKING_SENSOR_DETECTED;
					END_IF					
				E_AutoStore_States.TRANSFER_WORKING_SENSOR_DETECTED:
					IF sensor_transfer_atWorkingPos OR TRUE THEN//todo:adjust the position
						eStates	:= E_AutoStore_States.LIFT_MOVE_UP;
					END_IF
					
				////////////////////////////lift move up///////////////////////////////////	
				E_AutoStore_States.LIFT_MOVE_UP:
					st_mcAxis_lift.mcMoveAbsolute.Execute	:= TRUE;					
					st_mcAxis_lift.rActualPosSet	:= rPos_lift_up;
					st_mcAxis_lift.rVelocitySet		:= 150;					
					IF st_mcAxis_lift.mcMoveAbsolute.Done THEN
						st_mcAxis_lift.mcMoveAbsolute.Execute	:= FALSE;
						eStates	:= E_AutoStore_States.DONE;
					END_IF		

				
				E_AutoStore_States.DONE:
					autostore_status	:= AutostoreStatus.READY;
					eStates	:= E_AutoStore_States.WAIT_CMD;
				E_AutoStore_States.ERROR:
					;
			END_CASE
		
		
	ePMLProtUnitMode_Maintenance, ePMLUnitMode_Service:		
		//
		
	ePMLProtUnitMode_Manual:		//Manaul

END_CASE
END_METHOD

{attribute 'object_name' := 'M_Holding'}
METHOD M_Holding
CASE fbUnitModeManager.eModeStatus OF
	ePMLProtUnitMode_Production:		//Mode Production
		//Finisch the actual seperationstep	
		

	ePMLProtUnitMode_Maintenance:
		M_StateComplete();
END_CASE
END_METHOD

{attribute 'object_name' := 'M_Idle'}
METHOD M_Idle
IF G_HMI.bAging_test THEN
	//M_agingTest();
END_IF
END_METHOD

METHOD M_mapping : BOOL
VAR_INPUT
END_VAR
IF sInstanceName='autoStore_1' THEN	
	(****************************digital input***************************************************)
	st_mcAxis_lift.limit_sensor_positive		:= 	arDI[20].Ch[0] ;
	st_mcAxis_lift.limit_sensor_negative		:= 	arDI[20].Ch[1] ;
	door_closed									:= 	arDI[20].Ch[2] ;
	button_start								:= 	arDI[20].Ch[3] ;
	button_stop									:= 	arDI[20].Ch[4] ;
	sensor_lift_atDownPos						:= 	arDI[20].Ch[5] ;
	st_mcAxis_transfer.limit_sensor_positive	:= 	arDI[20].Ch[6] ;
	st_mcAxis_transfer.limit_sensor_negative	:= 	arDI[20].Ch[7] ;	
	sensor_transfer_atWorkingPos				:= 	arDI[20].Ch[8] ;	
//	sensor_transfer_atFeedingPos				:= 	arDI[20].Ch[9] ;	
		

	/////////////////////////////////////axis config////////////////////////////////////////
	mcAxis_transfer
	(
		ZSN		:=  TRUE OR (st_mcAxis_transfer.limit_sensor_negative (*AND sensor_lift_atDownPos*)) OR st_mcAxis_transfer.xHoming, //TODO link to digital input
		ZSP		:=  TRUE OR (st_mcAxis_transfer.limit_sensor_positive (*AND sensor_lift_atDownPos*)) OR st_mcAxis_transfer.xHoming, //TODO link to digital input
		IN_OUT	:= st_mcAxis_transfer	, 
		AXIS	:= AxisRef_transfer	, 
	);
	st_mcAxis_transfer.bPosSensorShow	:= TRUE;
	st_mcAxis_transfer.bNegSensorShow	:= TRUE;
	st_mcAxis_transfer.bStopButtonShow	:= TRUE;
	st_mcAxis_transfer.rMaxAcceleration	:= 50000;
	st_mcAxis_transfer.rMaxDeceleration	:= 50000;
	st_mcAxis_transfer.rMaxJerk			:= 500000;
	st_mcAxis_transfer.rAcceleration	:= 2500;
	st_mcAxis_transfer.rDeceleration	:= 2500;
	st_mcAxis_transfer.rJerk			:= 12500;
	st_mcAxis_transfer.rMaxVelocity		:= 100;
	st_mcAxis_transfer.rMaxDistance		:= 50;
	st_mcAxis_transfer.bPosSen	:=  st_mcAxis_transfer.limit_sensor_positive ;//TODO link to digital input
	st_mcAxis_transfer.bNegSen	:=  st_mcAxis_transfer.limit_sensor_negative ;//TODO link to digital input
	st_mcAxis_transfer.mcHome.bCalibrationCam	:= TRUE;//TODO link to digital input origin
	st_mcAxis_transfer.bPositionSensor	:= TRUE;//TODO link to digital input origin
	st_mcAxis_transfer.bdirFW	:= TRUE;
	st_mcAxis_transfer.sNetID := '192.168.11.159.8.1';
	st_mcAxis_transfer.nSlaveAddr	:= 1004;
	st_mcAxis_transfer.rToqueLimitSet	:= 80;	
	
	mcAxis_lift
	(
		ZSN		:=   TRUE OR st_mcAxis_lift.limit_sensor_negative  OR st_mcAxis_lift.xHoming, //TODO link to digital input
		ZSP		:=   TRUE OR (st_mcAxis_lift.limit_sensor_positive (*AND sensor_transfer_atWorkingPos*))  OR st_mcAxis_lift.xHoming, //TODO link to digital input
		IN_OUT	:= st_mcAxis_lift	, 
		AXIS	:= AxisRef_lift	, 
	);
	st_mcAxis_lift.bPosSensorShow	:= TRUE;
	st_mcAxis_lift.bNegSensorShow	:= TRUE;
	st_mcAxis_lift.bStopButtonShow	:= TRUE;
	st_mcAxis_lift.rMaxAcceleration	:= 50000;
	st_mcAxis_lift.rMaxDeceleration	:= 50000;
	st_mcAxis_lift.rMaxJerk			:= 500000;
	st_mcAxis_lift.rAcceleration	:= 2500;
	st_mcAxis_lift.rDeceleration	:= 2500;
	st_mcAxis_lift.rJerk			:= 12500;
	st_mcAxis_lift.rMaxVelocity		:= 100;
	st_mcAxis_lift.rMaxDistance		:= 50;
	st_mcAxis_lift.bPosSen	:=  st_mcAxis_lift.limit_sensor_positive ;//TODO link to digital input
	st_mcAxis_lift.bNegSen	:=  TRUE(*st_mcAxis_lift.limit_sensor_negative*) ;//TODO link to digital input
	st_mcAxis_lift.mcHome.bCalibrationCam	:= TRUE;//TODO link to digital input origin
	st_mcAxis_lift.bPositionSensor	:= TRUE;//TODO link to digital input origin
	st_mcAxis_lift.bdirFW	:= TRUE;
	st_mcAxis_lift.sNetID := '192.168.11.159.8.1';
	st_mcAxis_lift.nSlaveAddr	:= 1005;
	st_mcAxis_lift.rToqueLimitSet	:= 80;
END_IF




IF sInstanceName='autoStore_2' THEN	
	(****************************digital input***************************************************)
	st_mcAxis_lift.limit_sensor_positive		:= 	arDI[21].Ch[0] ;
	st_mcAxis_lift.limit_sensor_negative		:= 	arDI[21].Ch[1] ;
	door_closed									:= 	arDI[21].Ch[2] ;
	button_start								:= 	arDI[21].Ch[3] ;
	button_stop									:= 	arDI[21].Ch[4] ;
	sensor_lift_atDownPos						:= 	arDI[21].Ch[5] ;
	st_mcAxis_transfer.limit_sensor_positive	:= 	arDI[21].Ch[6] ;
	st_mcAxis_transfer.limit_sensor_negative	:= 	arDI[21].Ch[7] ;	
	sensor_transfer_atWorkingPos				:= 	arDI[21].Ch[8] ;	
//	sensor_transfer_atFeedingPos				:= 	arDI[21].Ch[9] ;	
		

	/////////////////////////////////////axis config////////////////////////////////////////
	mcAxis_transfer
	(
		ZSN		:=  TRUE OR (st_mcAxis_transfer.limit_sensor_negative (*AND sensor_lift_atDownPos*)) OR st_mcAxis_transfer.xHoming, //TODO link to digital input
		ZSP		:=  TRUE OR (st_mcAxis_transfer.limit_sensor_positive (*AND sensor_lift_atDownPos*)) OR st_mcAxis_transfer.xHoming, //TODO link to digital input
		IN_OUT	:= st_mcAxis_transfer	, 
		AXIS	:= AxisRef_transfer	, 
	);
	st_mcAxis_transfer.bPosSensorShow	:= TRUE;
	st_mcAxis_transfer.bNegSensorShow	:= TRUE;
	st_mcAxis_transfer.bStopButtonShow	:= TRUE;
	st_mcAxis_transfer.rMaxAcceleration	:= 50000;
	st_mcAxis_transfer.rMaxDeceleration	:= 50000;
	st_mcAxis_transfer.rMaxJerk			:= 500000;
	st_mcAxis_transfer.rAcceleration	:= 2500;
	st_mcAxis_transfer.rDeceleration	:= 2500;
	st_mcAxis_transfer.rJerk			:= 12500;
	st_mcAxis_transfer.rMaxVelocity		:= 100;
	st_mcAxis_transfer.rMaxDistance		:= 50;
	st_mcAxis_transfer.bPosSen	:=  st_mcAxis_transfer.limit_sensor_positive ;//TODO link to digital input
	st_mcAxis_transfer.bNegSen	:=  st_mcAxis_transfer.limit_sensor_negative ;//TODO link to digital input
	st_mcAxis_transfer.mcHome.bCalibrationCam	:= TRUE;//TODO link to digital input origin
	st_mcAxis_transfer.bPositionSensor	:= TRUE;//TODO link to digital input origin
	st_mcAxis_transfer.bdirFW	:= TRUE;
	st_mcAxis_transfer.sNetID := '192.168.11.159.10.1';
	st_mcAxis_transfer.nSlaveAddr	:= 1004;
	st_mcAxis_transfer.rToqueLimitSet	:= 80;	
	
	mcAxis_lift
	(
		ZSN		:=   TRUE OR st_mcAxis_lift.limit_sensor_negative  OR st_mcAxis_lift.xHoming, //TODO link to digital input
		ZSP		:=   TRUE OR (st_mcAxis_lift.limit_sensor_positive (*AND sensor_transfer_atWorkingPos*))  OR st_mcAxis_lift.xHoming, //TODO link to digital input
		IN_OUT	:= st_mcAxis_lift	, 
		AXIS	:= AxisRef_lift	, 
	);
	st_mcAxis_lift.bPosSensorShow	:= TRUE;
	st_mcAxis_lift.bNegSensorShow	:= TRUE;
	st_mcAxis_lift.bStopButtonShow	:= TRUE;
	st_mcAxis_lift.rMaxAcceleration	:= 50000;
	st_mcAxis_lift.rMaxDeceleration	:= 50000;
	st_mcAxis_lift.rMaxJerk			:= 500000;
	st_mcAxis_lift.rAcceleration	:= 2500;
	st_mcAxis_lift.rDeceleration	:= 2500;
	st_mcAxis_lift.rJerk			:= 12500;
	st_mcAxis_lift.rMaxVelocity		:= 100;
	st_mcAxis_lift.rMaxDistance		:= 50;
	st_mcAxis_lift.bPosSen	:=  st_mcAxis_lift.limit_sensor_positive ;//TODO link to digital input
	st_mcAxis_lift.bNegSen	:=  TRUE(*st_mcAxis_lift.limit_sensor_negative*) ;//TODO link to digital input
	st_mcAxis_lift.mcHome.bCalibrationCam	:= TRUE;//TODO link to digital input origin
	st_mcAxis_lift.bPositionSensor	:= TRUE;//TODO link to digital input origin
	st_mcAxis_lift.bdirFW	:= TRUE;
	st_mcAxis_lift.sNetID := '192.168.11.159.10.1';
	st_mcAxis_lift.nSlaveAddr	:= 1005;
	st_mcAxis_lift.rToqueLimitSet	:= 80;
END_IF
END_METHOD

METHOD M_Reset
VAR_INPUT
END_VAR
//Take away all commands
IF GVL.stChangeIntoProduction.bYesReset THEN
;
END_IF
END_METHOD

{attribute 'object_name' := 'M_Resetting'}
METHOD M_Resetting
CASE fbUnitModeManager.eModeStatus OF
	ePMLProtUnitMode_Production:		//Production, Mantainance, Manual
		lamp	:= FALSE;
		eStates :=E_SampleStates.IDLE;
		M_StateComplete();
	
	ePMLProtUnitMode_Maintenance, ePMLProtUnitMode_Manual, ePMLUnitMode_Service:
		M_StateComplete();
END_CASE
END_METHOD

{attribute 'object_name' := 'M_Starting'}
METHOD M_Starting
CASE fbUnitModeManager.eModeStatus OF
	ePMLProtUnitMode_Production:		//Production, Mantainance, Manual
		st_mcAxis_transfer.mcPower.Enable	:= TRUE;
		st_mcAxis_lift.mcPower.Enable	:= TRUE;
		IF st_mcAxis_transfer.mcPower.Status AND st_mcAxis_lift.mcPower.Status THEN
			eStates	:= E_AutoStore_States.IDLE;	
			M_StateComplete();
		END_IF
		
	ePMLProtUnitMode_Maintenance, ePMLProtUnitMode_Manual, ePMLUnitMode_Service:
		M_StateComplete();
END_CASE
END_METHOD

{attribute 'object_name' := 'M_Stopping'}
METHOD M_Stopping

CASE fbUnitModeManager.eModeStatus OF
	ePMLProtUnitMode_Production:		//Mode Production
//////////////////////////////////////////////////////////timeout//////////////////////////////////////////	
		iStateTemp	:= eStateTemp;
		ton_timeout();
		IF eStateTemp=eStates THEN
			ton_timeout.IN	:=TRUE;
		ELSE
			ton_timeout.IN	:=FALSE;
			eStateTemp	:= eStates;	
			M_Log(eLogType:=ServerityLevelType.INFO,sTextLog:='');
			IF ton_timeout.Q THEN
				RETURN;
			END_IF
		END_IF
		IF ton_timeout.Q THEN	
			ton_timeout.IN	:=FALSE;
			CASE eStates OF	
				E_AutoStore_States.ERROR:	
					alarm_temp.Message	:= GenerateErrorMsg(errorType:='M',iState := iStateTemp,errorMsg:='in error state.');
				ELSE
				alarm_temp.Message	:= GenerateErrorMsg(errorType:='M',iState := iStateTemp,errorMsg:='time out');
			END_CASE
//////////////////////////////////////////////////////////states don't want to timeout and trig error//////////////////////////////////////////				
			IF 	eStates<>E_AutoStore_States.IDLE AND
				eStates<>E_AutoStore_States.WAIT AND
				eStates<>E_AutoStore_States.WAIT_CMD
			THEN 
				IF sInstanceName='autoStore_1' THEN
					GVL.pml_adminAlarm.M_SetAlarm(stAdmin:=GVL.PackTags1.Admin,stAlarm:=alarm_temp);
				END_IF
				IF sInstanceName='autoStore_2' THEN
					GVL.pml_adminAlarm.M_SetAlarm(stAdmin:=GVL.PackTags2.Admin,stAlarm:=alarm_temp);
				END_IF					
			END_IF
		END_IF
//////////////////////////////////////////////////////////auto running process//////////////////////////////////////////			
		CASE eStates OF 
				E_AutoStore_States.IDLE:
					ton_timeout.PT	:= T#1MS;						
					eStates	:= E_AutoStore_States.INIT;				
				E_AutoStore_States.INIT:
					ton_timeout.PT	:= T#1S;
					eStates	:= E_AutoStore_States.WAIT; 
				E_AutoStore_States.WAIT:
					ton_timeout.PT	:= T#10S;
					eStates	:= E_AutoStore_States.WAIT_CMD; 
				E_AutoStore_States.WAIT_CMD:
					M_StateComplete();
					IF bExchangeTote THEN
						bExchangeTote	:= FALSE;
						eStates	:= E_AutoStore_States.LIFT_MOVE_DOWN;
					END_IF
				////////////////////////////lift move down///////////////////////////////////		
				E_AutoStore_States.LIFT_MOVE_DOWN:	
					st_mcAxis_lift.mcMoveAbsolute.Execute	:= TRUE;					
					st_mcAxis_lift.rActualPosSet	:= rPos_lift_down;
					st_mcAxis_lift.rVelocitySet		:= 100;					
					IF st_mcAxis_lift.mcMoveAbsolute.Done THEN
						eStates	:= E_AutoStore_States.LIFT_DOWN_SENSOR_DETECTED;
					END_IF
				E_AutoStore_States.LIFT_DOWN_SENSOR_DETECTED:	
					IF sensor_lift_atDownPos THEN
						IF bUpStairs THEN
							eStates	:= E_AutoStore_States.TRANSFER_MOVE_FEEDING;
							bUpStairs	:= FALSE;
						ELSE
							eStates	:= E_AutoStore_States.TRANSFER_MOVE_WORKING;
							bUpStairs	:= TRUE;
						END_IF					
					END_IF
				////////////////////////////upstairs///////////////////////////////////	
				E_AutoStore_States.TRANSFER_MOVE_FEEDING:	
					st_mcAxis_transfer.mcMoveAbsolute.Execute	:= TRUE;					
					st_mcAxis_transfer.rActualPosSet	:= rPos_transfer_feeding;
					st_mcAxis_transfer.rVelocitySet		:= 100;					
					IF st_mcAxis_transfer.mcMoveAbsolute.Done THEN
						eStates	:= E_AutoStore_States.TRANSFER_FEEDING_SENSOR_DETECTED;
					END_IF				

				E_AutoStore_States.TRANSFER_FEEDING_SENSOR_DETECTED:
					IF sensor_transfer_atFeedingPos OR TRUE THEN//todo:add this sensor
						eStates	:= E_AutoStore_States.LIFT_MOVE_UP;
					END_IF									
				////////////////////////////downstairs///////////////////////////////////		
				E_AutoStore_States.TRANSFER_MOVE_WORKING:	
					st_mcAxis_transfer.mcMoveAbsolute.Execute	:= TRUE;					
					st_mcAxis_transfer.rActualPosSet	:= rPos_transfer_working;
					st_mcAxis_transfer.rVelocitySet		:= 100;					
					IF st_mcAxis_transfer.mcMoveAbsolute.Done THEN
						eStates	:= E_AutoStore_States.TRANSFER_WORKING_SENSOR_DETECTED;
					END_IF					
				E_AutoStore_States.TRANSFER_WORKING_SENSOR_DETECTED:
					IF sensor_transfer_atWorkingPos THEN
						eStates	:= E_AutoStore_States.LIFT_MOVE_UP;
					END_IF
					
				////////////////////////////lift move up///////////////////////////////////	
				E_AutoStore_States.LIFT_MOVE_UP:
					st_mcAxis_lift.mcMoveAbsolute.Execute	:= TRUE;					
					st_mcAxis_lift.rActualPosSet	:= rPos_lift_up;
					st_mcAxis_lift.rVelocitySet		:= 100;					
					IF st_mcAxis_lift.mcMoveAbsolute.Done THEN
						eStates	:= E_AutoStore_States.DONE;
					END_IF		

				
				E_AutoStore_States.DONE:
					eStates	:= E_AutoStore_States.IDLE;
					M_StateComplete();
				E_AutoStore_States.ERROR:
					;
			END_CASE
		
		
	ePMLProtUnitMode_Maintenance, ePMLUnitMode_Service:		
		//
		
	ePMLProtUnitMode_Manual:		//Manaul

END_CASE
END_METHOD

{attribute 'object_name' := 'M_Undefined'}
METHOD M_Undefined

bUndefinedDone					:= TRUE;
END_METHOD

METHOD ParseStateToString : STRING
VAR_INPUT
END_VAR
CASE THIS^.eStates OF
	E_AutoStore_States.IDLE:
		ParseStateToString	:='IDLE';
	E_AutoStore_States.INIT:
		ParseStateToString	:='INIT';
	E_AutoStore_States.CHECK:
		ParseStateToString	:='CHECK';

	E_AutoStore_States.WAIT:
		ParseStateToString	:='WAIT';

	E_AutoStore_States.DONE:	
		ParseStateToString	:='DONE';
	E_AutoStore_States.ERROR:
		ParseStateToString	:='ERROR';
	ELSE
		ParseStateToString	:='UNKNOW STATE';
END_CASE
END_METHOD

END_FUNCTION_BLOCK

// ---- Mian/FB_working_tote.TcPOU
FUNCTION_BLOCK FB_working_tote EXTENDS FB_Generic
VAR_IN_OUT
	
END_VAR
VAR_INPUT
	
END_VAR
VAR_OUTPUT
	error_status	: OrderToteErrorStatus := OrderToteErrorStatus.UNKNOWN;	
	bag_opening_status	:ARRAY[0..1]OF BagOpeningStatus;
END_VAR
VAR
	eStates				: E_WorkingStates	:= E_WorkingStates.IDLE;
	eStateTemp			: E_WorkingStates	:= E_WorkingStates.IDLE;
	tote_status			: ToteStatus;
	outboundTote_status	: ToteStatus;
	

//	bag_opening_status_0	: REFERENCE TO BagOpeningStatus;
//	bag_opening_status_1	: REFERENCE TO BagOpeningStatus;
	bagOpen_Status			: ARRAY[0..1] OF ST_BagOpen;
	bagOpenInit_Status		: ARRAY[0..1] OF ST_BagOpen;
	
	iCount_sensor_detection	: ARRAY [0..1] OF INT;
	strLog_bagopen_detection	: STRING;
	
//	bOpen_bag_detection		: BOOL	:= TRUE;
//	bOpen_bag_detection_0	: BOOL	:= TRUE;
//	bOpen_bag_detection_1	: BOOL	:= TRUE;
	
	logtech_control_command	: LogTechControlCmd;
	logtech_status	:LogTechStatus;
	logtech_transfer_status	: LogTechTransferStatus;
	//rPos_bag_closed_step_0	: REAL;  //半开袋位置设定
	bRobot_in_safety_place	: BOOL:=TRUE;
///////

	valve_lift			: Valve;
	roller_preInbound	: Roller;
	roller_inbound		: Inbound;
	roller_outbound		: Outbound;
	roller_outbound_assist	: Outbound;
	
	photo_sensor_tote_detection: FB_DigitalInput;
	
    BagOpening_Detection	: ARRAY[0..7] OF BOOL;
	sensor_cover			: ARRAY[0..1] OF BOOL;
	EDM_KM			    : BOOL;
	
	mcAxis_lift 		: FB_MotionAxis_MC;
	st_mcAxis_lift 		: ST_MotionAxis_MC;
	AxisRef_lift		: AXIS_REF;
	
	mcAxis_bag 			: FB_MotionAxis_MC;
	st_mcAxis_bag		: ST_MotionAxis_MC;
	AxisRef_bag			: AXIS_REF;		
	
//	xLoading : BOOL;
//	xUnloading : BOOL;
	xInbound	: BOOL;
	xOutbound	: BOOL;
	rPos_bag_closed_step_0	: REAL;
	
	
	xBeginInbound	: BOOL;
	xAbortInbound	: BOOL;
	xAbortOutbound	: BOOL;
	
	rTrig1	: R_TRIG;
	fTrig1	: F_TRIG;
	str4debug	: STRING;
	eState_temp1	: STRING;
	state_track		: STRING(255);
	
	
	
	stSubModuleInfo		: ARRAY [1..iSubModule] OF ST_PMLSubUnitInfo;	//Informations about the Subunits
	bMachineStartedUp	: BOOL;
	eCommand_manual		: E_PMLCommand;
END_VAR

VAR CONSTANT
	rMax_lift	: REAL	:= 135;
	rMin_lift	: REAL	:= -0.5;
	rMax_bag	: REAL	:= 56;
	rMin_bag	: REAL	:= -0.5;	
	
	iSubModule		: UDINT:=1;
END_VAR

VAR PERSISTENT
	rPos_lift_up				: REAL;
	rPos_lift_down				: REAL;
	rPos_bag_opened				: REAL;
	rPos_bag_closed				: REAL;	
	rPos_bag_preopen			: REAL;
	iDelay_sensor_detection		: INT;
	iSensor_detection_setting	: ARRAY [0..1] OF INT;
	bUsingOpenBag				: BOOL;
END_VAR

SUPER^();
infoLevel	:= ServerityLevelType.WARNING;
IF sInstanceName='working1' THEN
	IF NOT subscribed THEN
		GVL.PubSubService.Subscribe(E_Topics.WORKING1_INBOUND_TOTE,sInstanceName,THIS^);
		GVL.PubSubService.Subscribe(E_Topics.WORKING1_OUTBOUND_TOTE,sInstanceName,THIS^);
		GVL.PubSubService.Subscribe(E_Topics.WORKING1_BEGIN_INBOUND,sInstanceName,THIS^);
		GVL.PubSubService.Subscribe(E_Topics.WORKING1_ABORT_INBOUND,sInstanceName,THIS^);
		GVL.PubSubService.Subscribe(E_Topics.WORKING1_ABORT_OUTBOUND,sInstanceName,THIS^);
		subscribed	:= TRUE;
	END_IF
END_IF
IF sInstanceName='working2' THEN
	IF NOT subscribed THEN
		GVL.PubSubService.Subscribe(E_Topics.WORKING2_INBOUND_TOTE,sInstanceName,THIS^);
		GVL.PubSubService.Subscribe(E_Topics.WORKING2_OUTBOUND_TOTE,sInstanceName,THIS^);	
		GVL.PubSubService.Subscribe(E_Topics.WORKING2_BEGIN_INBOUND,sInstanceName,THIS^);
		GVL.PubSubService.Subscribe(E_Topics.WORKING2_ABORT_INBOUND,sInstanceName,THIS^);
		GVL.PubSubService.Subscribe(E_Topics.WORKING2_ABORT_OUTBOUND,sInstanceName,THIS^);

		subscribed	:= TRUE;
	END_IF
END_IF


//bag_opening_status_0	REF= MAIN.tote_1.working1_tote.bag_opening_status_0;
//bag_opening_status_1	REF= MAIN.tote_1.working2_tote.bag_opening_status_1;

bagOpenInit_Status[0].bag_status				:=BagStatus.UNOPENED;
bagOpenInit_Status[0].iCnt_sensor_detection		:=0;
bagOpenInit_Status[0].sensor_status				:='';
bagOpenInit_Status[1].bag_status				:=BagStatus.UNOPENED;
bagOpenInit_Status[1].iCnt_sensor_detection		:=0;
bagOpenInit_Status[1].sensor_status				:='';
////////////////////////////////////////////////mechanical error///////////////////////////////////////////////////
IF GVL.fb_loading.tote_status=ToteStatus.MECHANICAL_ERROR THEN
	tote_status	:= ToteStatus.MECHANICAL_ERROR;
END_IF
////////////////////////////////////////////////electrical error///////////////////////////////////////////////////
rTrig_electricalError[1](CLK:= st_mcAxis_lift.mcReadStatus.Error);
rTrig_electricalError[2](CLK:= st_mcAxis_bag.mcReadStatus.Error);
rTrig_electricalError[3](CLK:= roller_inbound.roller.err.Q);
rTrig_electricalError[4](CLK:= roller_outbound.roller.err.Q);
rTrig_electricalError[5](CLK:= roller_outbound_assist.roller.err.Q);
IF sInstanceName='working1' THEN
	IF GVL.PackTags1.Status.StateCurrent<>E_PMLState.ePMLState_Resetting THEN
		FOR i:=1 TO 10 DO
			IF rTrig_electricalError[i].Q THEN
				THIS^.packTags.Admin.Alarm[i].ID	:= i;
				CASE i OF
					1:
						THIS^.packTags.Admin.Alarm[1].Message	:= GenerateErrorMsg(errorType:='E',iState := i,errorMsg:='lift axis is in error state.');
					2:
						THIS^.packTags.Admin.Alarm[2].Message	:= GenerateErrorMsg(errorType:='E',iState := i,errorMsg:='open bag axis of working is in error state.');
					3:
						THIS^.packTags.Admin.Alarm[3].Message	:= GenerateErrorMsg(errorType:='E',iState := i,errorMsg:='inbound roller is in error state.');
					4:
						THIS^.packTags.Admin.Alarm[4].Message	:= GenerateErrorMsg(errorType:='E',iState := i,errorMsg:='outbound roller is in error state.');
					5:
						THIS^.packTags.Admin.Alarm[5].Message	:= GenerateErrorMsg(errorType:='E',iState := i,errorMsg:='outbound assist roller is in error state.');
				END_CASE
					tote_status	:= ToteStatus.ELECTRICAL_ERROR;
					GVL.pml_adminAlarm.M_SetAlarm(stAdmin:=GVL.PackTags1.Admin,stAlarm := THIS^.packTags.Admin.Alarm[i]);			
			END_IF
		END_FOR
	END_IF	
END_IF
IF sInstanceName='working2' THEN
	IF GVL.PackTags2.Status.StateCurrent<>E_PMLState.ePMLState_Resetting THEN
		FOR i:=1 TO 10 DO
			IF rTrig_electricalError[i].Q THEN
				THIS^.packTags.Admin.Alarm[i].ID	:= i;
				CASE i OF
					1:
						THIS^.packTags.Admin.Alarm[1].Message	:= GenerateErrorMsg(errorType:='E',iState := i,errorMsg:='lift axis is in error state.');
					2:
						THIS^.packTags.Admin.Alarm[2].Message	:= GenerateErrorMsg(errorType:='E',iState := i,errorMsg:='open bag axis of working is in error state.');
					3:
						THIS^.packTags.Admin.Alarm[3].Message	:= GenerateErrorMsg(errorType:='E',iState := i,errorMsg:='inbound roller is in error state.');
					4:
						THIS^.packTags.Admin.Alarm[4].Message	:= GenerateErrorMsg(errorType:='E',iState := i,errorMsg:='outbound roller is in error state.');
					5:
						THIS^.packTags.Admin.Alarm[5].Message	:= GenerateErrorMsg(errorType:='E',iState := i,errorMsg:='outbound assist roller is in error state.');
				END_CASE	
				GVL.pml_adminAlarm.M_SetAlarm(stAdmin:=GVL.PackTags2.Admin,stAlarm := THIS^.packTags.Admin.Alarm[i]);			
			END_IF
		END_FOR
	END_IF	
END_IF


